LIN {X 103.200,Y -21.699,Z -137.911,A -90.000,B 90.000,C 0.000} C_DIS
LIN {X 103.154,Y -21.706,Z -138.831,A -90.000,B 90.000,C 0.000} C_DIS
LIN {X 102.985,Y -21.715,Z -141.880,A -90.000,B 90.000,C 0.000} C_DIS
LIN {X 102.956,Y -21.718,Z -142.349,A -90.000,B 90.000,C 0.000} C_DIS
LIN {X 102.711,Y -21.728,Z -146.129,A -90.000,B 90.000,C 0.000} C_DIS
LIN {X 102.478,Y -21.737,Z -149.340,A -90.000,B 90.000,C 0.000} C_DIS
LIN {X 102.272,Y -21.746,Z -151.898,A -90.000,B 90.000,C 0.000} C_DIS
LIN {X 102.195,Y -21.747,Z -152.952,A -90.000,B 90.000,C 0.000} C_DIS
LIN {X 102.172,Y -21.748,Z -153.237,A -90.000,B 90.000,C 0.000} C_DIS
LIN {X 101.990,Y -21.757,Z -155.321,A -90.000,B 90.000,C 0.000} C_DIS
LIN {X 101.952,Y -21.757,Z -155.803,A -90.000,B 90.000,C 0.000} C_DIS
LIN {X 101.875,Y -21.759,Z -156.808,A -90.000,B 90.000,C 0.000} C_DIS
LIN {X 101.833,Y -21.759,Z -157.268,A -90.000,B 90.000,C 0.000} C_DIS
LIN {X 101.694,Y -21.768,Z -158.747,A -90.000,B 90.000,C 0.000} C_DIS
LIN {X 101.636,Y -21.768,Z -159.458,A -90.000,B 90.000,C 0.000} C_DIS
LIN {X 101.552,Y -21.770,Z -160.519,A -90.000,B 90.000,C 0.000} C_DIS
LIN {X 101.526,Y -21.769,Z -160.801,A -90.000,B 90.000,C 0.000} C_DIS
LIN {X 101.473,Y -21.773,Z -161.328,A -90.000,B 90.000,C 0.000} C_DIS
LIN {X 101.406,Y -21.769,Z -162.061,A -90.000,B 90.000,C 0.000} C_DIS
LIN {X 101.227,Y -21.773,Z -164.255,A -90.000,B 90.000,C 0.000} C_DIS
LIN {X 101.195,Y -21.774,Z -164.609,A -90.000,B 90.000,C 0.000} C_DIS
LIN {X 101.168,Y -21.773,Z -164.885,A -90.000,B 90.000,C 0.000} C_DIS
LIN {X 100.874,Y -21.791,Z -168.265,A -90.000,B 90.000,C 0.000} C_DIS
LIN {X 100.554,Y -21.808,Z -171.701,A -90.000,B 90.000,C 0.000} C_DIS
LIN {X 100.400,Y -21.816,Z -173.250,A -90.000,B 90.000,C 0.000} C_DIS
LIN {X 100.226,Y -21.828,Z -174.986,A -90.000,B 90.000,C 0.000} C_DIS
LIN {X 100.198,Y -21.826,Z -175.266,A -90.000,B 90.000,C 0.000} C_DIS
LIN {X 99.941,Y -21.835,Z -177.681,A -90.000,B 90.000,C 0.000} C_DIS
LIN {X 99.892,Y -21.832,Z -178.165,A -90.000,B 90.000,C 0.000} C_DIS
LIN {X 99.862,Y -21.833,Z -178.432,A -90.000,B 90.000,C 0.000} C_DIS
LIN {X 99.723,Y -21.828,Z -179.586,A -90.000,B 90.000,C 0.000} C_DIS
LIN {X 99.550,Y -21.810,Z -181.085,A -90.000,B 90.000,C 0.000} C_DIS
LIN {X 99.434,Y -21.803,Z -182.000,A -90.000,B 90.000,C 0.000} C_DIS
LIN {X 99.202,Y -21.777,Z -183.867,A -90.000,B 90.000,C 0.000} C_DIS
LIN {X 99.146,Y -21.771,Z -184.282,A -90.000,B 90.000,C 0.000} C_DIS
LIN {X 98.820,Y -21.726,Z -186.729,A -90.000,B 90.000,C 0.000} C_DIS
LIN {X 98.551,Y -21.689,Z -188.733,A -90.000,B 90.000,C 0.000} C_DIS
LIN {X 98.240,Y -21.655,Z -191.111,A -90.000,B 90.000,C 0.000} C_DIS
LIN {X 98.078,Y -21.642,Z -192.230,A -90.000,B 90.000,C 0.000} C_DIS
LIN {X 97.900,Y -21.626,Z -193.439,A -90.000,B 90.000,C 0.000} C_DIS
LIN {X 97.865,Y -21.625,Z -193.671,A -90.000,B 90.000,C 0.000} C_DIS
LIN {X 97.839,Y -21.622,Z -193.828,A -90.000,B 90.000,C 0.000} C_DIS
LIN {X 97.584,Y -21.620,Z -195.289,A -90.000,B 90.000,C 0.000} C_DIS
LIN {X 97.330,Y -21.612,Z -196.692,A -90.000,B 90.000,C 0.000} C_DIS
LIN {X 97.302,Y -21.611,Z -196.843,A -90.000,B 90.000,C 0.000} C_DIS
LIN {X 97.260,Y -21.612,Z -197.057,A -90.000,B 90.000,C 0.000} C_DIS
LIN {X 96.796,Y -21.616,Z -199.323,A -90.000,B 90.000,C 0.000} C_DIS
LIN {X 96.529,Y -21.612,Z -200.569,A -90.000,B 90.000,C 0.000} C_DIS
LIN {X 96.463,Y -21.611,Z -200.859,A -90.000,B 90.000,C 0.000} C_DIS
LIN {X 95.804,Y -21.631,Z -203.660,A -90.000,B 90.000,C 0.000} C_DIS
LIN {X 95.494,Y -21.634,Z -204.941,A -90.000,B 90.000,C 0.000} C_DIS
LIN {X 95.323,Y -21.635,Z -205.637,A -90.000,B 90.000,C 0.000} C_DIS
LIN {X 94.278,Y -21.666,Z -209.816,A -90.000,B 90.000,C 0.000} C_DIS
LIN {X 93.985,Y -21.666,Z -210.965,A -90.000,B 90.000,C 0.000} C_DIS
LIN {X 92.877,Y -21.692,Z -215.251,A -90.000,B 90.000,C 0.000} C_DIS
LIN {X 92.712,Y -21.692,Z -215.887,A -90.000,B 90.000,C 0.000} C_DIS
LIN {X 92.490,Y -21.690,Z -216.750,A -90.000,B 90.000,C 0.000} C_DIS
LIN {X 91.455,Y -21.706,Z -220.703,A -90.000,B 90.000,C 0.000} C_DIS
LIN {X 90.619,Y -21.709,Z -223.906,A -90.000,B 90.000,C 0.000} C_DIS
LIN {X 90.094,Y -21.704,Z -225.931,A -90.000,B 90.000,C 0.000} C_DIS
LIN {X 90.051,Y -21.703,Z -226.091,A -90.000,B 90.000,C 0.000} C_DIS
LIN {X 89.413,Y -21.699,Z -228.410,A -90.000,B 90.000,C 0.000} C_DIS
LIN {X 88.561,Y -21.691,Z -231.519,A -90.000,B 90.000,C 0.000} C_DIS
LIN {X 88.509,Y -21.688,Z -231.694,A -90.000,B 90.000,C 0.000} C_DIS
LIN {X 87.993,Y -21.687,Z -233.408,A -90.000,B 90.000,C 0.000} C_DIS
LIN {X 86.773,Y -21.676,Z -237.465,A -90.000,B 90.000,C 0.000} C_DIS
LIN {X 86.686,Y -21.679,Z -237.741,A -90.000,B 90.000,C 0.000} C_DIS
LIN {X 86.213,Y -21.680,Z -239.140,A -90.000,B 90.000,C 0.000} C_DIS
LIN {X 85.045,Y -21.673,Z -242.614,A -90.000,B 90.000,C 0.000} C_DIS
LIN {X 84.730,Y -21.673,Z -243.561,A -90.000,B 90.000,C 0.000} C_DIS
LIN {X 84.730,Y -60.000,Z -243.561,A -90.000,B 90.000,C 0.000} C_DIS
LIN {X -106.254,Y -60.000,Z -243.561,A -90.000,B 90.000,C 0.000} C_DIS
LIN {X -106.254,Y -21.411,Z -243.561,A -90.000,B 90.000,C 0.000} C_DIS
LIN {X -105.827,Y -21.342,Z -243.259,A -90.000,B 90.000,C 0.000} C_DIS
LIN {X -103.067,Y -21.337,Z -241.434,A -90.000,B 90.000,C 0.000} C_DIS
LIN {X -99.700,Y -21.332,Z -239.239,A -90.000,B 90.000,C 0.000} C_DIS
LIN {X -95.248,Y -21.329,Z -236.322,A -90.000,B 90.000,C 0.000} C_DIS
LIN {X -91.046,Y -21.329,Z -233.611,A -90.000,B 90.000,C 0.000} C_DIS
LIN {X -87.083,Y -21.328,Z -231.061,A -90.000,B 90.000,C 0.000} C_DIS
LIN {X -82.491,Y -21.331,Z -228.162,A -90.000,B 90.000,C 0.000} C_DIS
LIN {X -81.014,Y -21.331,Z -227.236,A -90.000,B 90.000,C 0.000} C_DIS
LIN {X -78.594,Y -21.335,Z -225.697,A -90.000,B 90.000,C 0.000} C_DIS
LIN {X -73.982,Y -21.346,Z -222.839,A -90.000,B 90.000,C 0.000} C_DIS
LIN {X -71.749,Y -21.350,Z -221.468,A -90.000,B 90.000,C 0.000} C_DIS
LIN {X -69.686,Y -21.361,Z -220.171,A -90.000,B 90.000,C 0.000} C_DIS
LIN {X -66.193,Y -21.389,Z -217.992,A -90.000,B 90.000,C 0.000} C_DIS
LIN {X -62.248,Y -21.420,Z -215.563,A -90.000,B 90.000,C 0.000} C_DIS
LIN {X -59.889,Y -21.450,Z -214.098,A -90.000,B 90.000,C 0.000} C_DIS
LIN {X -57.151,Y -21.489,Z -212.404,A -90.000,B 90.000,C 0.000} C_DIS
LIN {X -54.976,Y -21.517,Z -211.076,A -90.000,B 90.000,C 0.000} C_DIS
LIN {X -54.531,Y -21.522,Z -210.805,A -90.000,B 90.000,C 0.000} C_DIS
LIN {X -53.089,Y -21.553,Z -209.900,A -90.000,B 90.000,C 0.000} C_DIS
LIN {X -52.244,Y -21.569,Z -209.368,A -90.000,B 90.000,C 0.000} C_DIS
LIN {X -49.132,Y -21.649,Z -207.418,A -90.000,B 90.000,C 0.000} C_DIS
LIN {X -47.972,Y -21.680,Z -206.695,A -90.000,B 90.000,C 0.000} C_DIS
LIN {X -46.144,Y -21.761,Z -205.510,A -90.000,B 90.000,C 0.000} C_DIS
LIN {X -43.428,Y -21.875,Z -203.761,A -90.000,B 90.000,C 0.000} C_DIS
LIN {X -42.555,Y -21.907,Z -203.192,A -90.000,B 90.000,C 0.000} C_DIS
LIN {X -40.956,Y -22.000,Z -202.120,A -90.000,B 90.000,C 0.000} C_DIS
LIN {X -40.168,Y -22.045,Z -201.596,A -90.000,B 90.000,C 0.000} C_DIS
LIN {X -38.826,Y -22.111,Z -200.682,A -90.000,B 90.000,C 0.000} C_DIS
LIN {X -38.138,Y -22.136,Z -200.199,A -90.000,B 90.000,C 0.000} C_DIS
LIN {X -37.944,Y -22.141,Z -200.056,A -90.000,B 90.000,C 0.000} C_DIS
LIN {X -37.389,Y -22.162,Z -199.640,A -90.000,B 90.000,C 0.000} C_DIS
LIN {X -36.329,Y -22.200,Z -198.837,A -90.000,B 90.000,C 0.000} C_DIS
LIN {X -34.180,Y -22.222,Z -197.104,A -90.000,B 90.000,C 0.000} C_DIS
LIN {X -33.953,Y -22.227,Z -196.919,A -90.000,B 90.000,C 0.000} C_DIS
LIN {X -32.090,Y -22.228,Z -195.331,A -90.000,B 90.000,C 0.000} C_DIS
LIN {X -30.755,Y -22.235,Z -194.205,A -90.000,B 90.000,C 0.000} C_DIS
LIN {X -30.074,Y -22.236,Z -193.626,A -90.000,B 90.000,C 0.000} C_DIS
LIN {X -27.945,Y -22.226,Z -191.825,A -90.000,B 90.000,C 0.000} C_DIS
LIN {X -27.695,Y -22.227,Z -191.609,A -90.000,B 90.000,C 0.000} C_DIS
LIN {X -27.149,Y -22.223,Z -191.131,A -90.000,B 90.000,C 0.000} C_DIS
LIN {X -25.105,Y -22.209,Z -189.370,A -90.000,B 90.000,C 0.000} C_DIS
LIN {X -24.930,Y -22.211,Z -189.215,A -90.000,B 90.000,C 0.000} C_DIS
LIN {X -24.541,Y -22.207,Z -188.853,A -90.000,B 90.000,C 0.000} C_DIS
LIN {X -22.451,Y -22.186,Z -186.958,A -90.000,B 90.000,C 0.000} C_DIS
LIN {X -22.349,Y -22.189,Z -186.862,A -90.000,B 90.000,C 0.000} C_DIS
LIN {X -21.597,Y -22.182,Z -186.102,A -90.000,B 90.000,C 0.000} C_DIS
LIN {X -19.952,Y -22.162,Z -184.488,A -90.000,B 90.000,C 0.000} C_DIS
LIN {X -19.814,Y -22.165,Z -184.348,A -90.000,B 90.000,C 0.000} C_DIS
LIN {X -18.083,Y -22.145,Z -182.471,A -90.000,B 90.000,C 0.000} C_DIS
LIN {X -17.843,Y -22.144,Z -182.206,A -90.000,B 90.000,C 0.000} C_DIS
LIN {X -17.415,Y -22.140,Z -181.731,A -90.000,B 90.000,C 0.000} C_DIS
LIN {X -17.370,Y -22.141,Z -181.681,A -90.000,B 90.000,C 0.000} C_DIS
LIN {X -15.624,Y -22.116,Z -179.571,A -90.000,B 90.000,C 0.000} C_DIS
LIN {X -15.250,Y -22.115,Z -179.111,A -90.000,B 90.000,C 0.000} C_DIS
LIN {X -15.094,Y -22.118,Z -178.911,A -90.000,B 90.000,C 0.000} C_DIS
LIN {X -13.181,Y -22.081,Z -176.292,A -90.000,B 90.000,C 0.000} C_DIS
LIN {X -13.050,Y -22.081,Z -176.110,A -90.000,B 90.000,C 0.000} C_DIS
LIN {X -12.917,Y -22.086,Z -175.919,A -90.000,B 90.000,C 0.000} C_DIS
LIN {X -11.259,Y -22.045,Z -173.288,A -90.000,B 90.000,C 0.000} C_DIS
LIN {X -11.080,Y -22.054,Z -172.984,A -90.000,B 90.000,C 0.000} C_DIS
LIN {X -11.024,Y -22.054,Z -172.881,A -90.000,B 90.000,C 0.000} C_DIS
LIN {X -9.686,Y -22.001,Z -170.299,A -90.000,B 90.000,C 0.000} C_DIS
LIN {X -9.547,Y -22.011,Z -170.002,A -90.000,B 90.000,C 0.000} C_DIS
LIN {X -8.642,Y -21.959,Z -167.714,A -90.000,B 90.000,C 0.000} C_DIS
LIN {X -8.538,Y -21.958,Z -167.438,A -90.000,B 90.000,C 0.000} C_DIS
LIN {X -8.445,Y -21.971,Z -167.158,A -90.000,B 90.000,C 0.000} C_DIS
LIN {X -8.313,Y -21.957,Z -166.630,A -90.000,B 90.000,C 0.000} C_DIS
LIN {X -7.867,Y -21.918,Z -164.877,A -90.000,B 90.000,C 0.000} C_DIS
LIN {X -7.834,Y -21.932,Z -164.681,A -90.000,B 90.000,C 0.000} C_DIS
LIN {X -7.719,Y -21.897,Z -163.007,A -90.000,B 90.000,C 0.000} C_DIS
LIN {X -7.727,Y -21.880,Z -162.907,A -90.000,B 90.000,C 0.000} C_DIS
LIN {X -7.905,Y -21.856,Z -162.077,A -90.000,B 90.000,C 0.000} C_DIS
LIN {X -7.916,Y -21.856,Z -162.021,A -90.000,B 90.000,C 0.000} C_DIS
LIN {X -7.996,Y -21.815,Z -161.796,A -90.000,B 90.000,C 0.000} C_DIS
LIN {X -8.060,Y -21.780,Z -161.607,A -90.000,B 90.000,C 0.000} C_DIS
LIN {X -8.241,Y -21.777,Z -161.247,A -90.000,B 90.000,C 0.000} C_DIS
LIN {X -8.444,Y -21.725,Z -160.934,A -90.000,B 90.000,C 0.000} C_DIS
LIN {X -8.526,Y -21.707,Z -160.802,A -90.000,B 90.000,C 0.000} C_DIS
LIN {X -8.552,Y -21.701,Z -160.759,A -90.000,B 90.000,C 0.000} C_DIS
LIN {X -8.873,Y -21.698,Z -160.372,A -90.000,B 90.000,C 0.000} C_DIS
LIN {X -8.932,Y -21.690,Z -160.309,A -90.000,B 90.000,C 0.000} C_DIS
LIN {X -9.104,Y -21.665,Z -160.116,A -90.000,B 90.000,C 0.000} C_DIS
LIN {X -9.212,Y -21.651,Z -159.991,A -90.000,B 90.000,C 0.000} C_DIS
LIN {X -9.330,Y -21.635,Z -159.850,A -90.000,B 90.000,C 0.000} C_DIS
LIN {X -9.669,Y -21.633,Z -159.535,A -90.000,B 90.000,C 0.000} C_DIS
LIN {X -9.815,Y -21.629,Z -159.394,A -90.000,B 90.000,C 0.000} C_DIS
LIN {X -10.168,Y -21.615,Z -159.041,A -90.000,B 90.000,C 0.000} C_DIS
LIN {X -10.408,Y -21.600,Z -158.806,A -90.000,B 90.000,C 0.000} C_DIS
LIN {X -11.277,Y -21.572,Z -158.006,A -90.000,B 90.000,C 0.000} C_DIS
LIN {X -11.496,Y -21.566,Z -157.804,A -90.000,B 90.000,C 0.000} C_DIS
LIN {X -11.881,Y -21.564,Z -157.468,A -90.000,B 90.000,C 0.000} C_DIS
LIN {X -13.335,Y -21.535,Z -156.177,A -90.000,B 90.000,C 0.000} C_DIS
LIN {X -13.574,Y -21.533,Z -155.965,A -90.000,B 90.000,C 0.000} C_DIS
LIN {X -15.277,Y -21.506,Z -154.485,A -90.000,B 90.000,C 0.000} C_DIS
LIN {X -15.775,Y -21.504,Z -154.059,A -90.000,B 90.000,C 0.000} C_DIS
LIN {X -17.794,Y -21.486,Z -152.333,A -90.000,B 90.000,C 0.000} C_DIS
LIN {X -18.467,Y -21.486,Z -151.758,A -90.000,B 90.000,C 0.000} C_DIS
LIN {X -20.638,Y -21.477,Z -149.908,A -90.000,B 90.000,C 0.000} C_DIS
LIN {X -20.734,Y -21.476,Z -149.825,A -90.000,B 90.000,C 0.000} C_DIS
LIN {X -20.875,Y -21.474,Z -149.698,A -90.000,B 90.000,C 0.000} C_DIS
LIN {X -23.951,Y -21.471,Z -146.908,A -90.000,B 90.000,C 0.000} C_DIS
LIN {X -24.114,Y -21.467,Z -146.745,A -90.000,B 90.000,C 0.000} C_DIS
LIN {X -27.216,Y -21.470,Z -143.581,A -90.000,B 90.000,C 0.000} C_DIS
LIN {X -27.540,Y -21.469,Z -143.244,A -90.000,B 90.000,C 0.000} C_DIS
LIN {X -27.679,Y -21.463,Z -143.078,A -90.000,B 90.000,C 0.000} C_DIS
LIN {X -29.860,Y -21.467,Z -140.414,A -90.000,B 90.000,C 0.000} C_DIS
LIN {X -30.541,Y -21.469,Z -139.579,A -90.000,B 90.000,C 0.000} C_DIS
LIN {X -30.827,Y -21.467,Z -139.209,A -90.000,B 90.000,C 0.000} C_DIS
LIN {X -31.012,Y -21.456,Z -138.921,A -90.000,B 90.000,C 0.000} C_DIS
LIN {X -32.519,Y -21.455,Z -136.513,A -90.000,B 90.000,C 0.000} C_DIS
LIN {X -33.305,Y -21.445,Z -135.260,A -90.000,B 90.000,C 0.000} C_DIS
LIN {X -33.469,Y -21.442,Z -134.995,A -90.000,B 90.000,C 0.000} C_DIS
LIN {X -33.552,Y -21.435,Z -134.865,A -90.000,B 90.000,C 0.000} C_DIS
LIN {X -33.811,Y -21.400,Z -134.386,A -90.000,B 90.000,C 0.000} C_DIS
LIN {X -34.144,Y -21.377,Z -133.751,A -90.000,B 90.000,C 0.000} C_DIS
LIN {X -34.605,Y -21.351,Z -132.868,A -90.000,B 90.000,C 0.000} C_DIS
LIN {X -35.010,Y -21.334,Z -132.094,A -90.000,B 90.000,C 0.000} C_DIS
LIN {X -35.479,Y -21.319,Z -131.192,A -90.000,B 90.000,C 0.000} C_DIS
LIN {X -35.801,Y -21.313,Z -130.570,A -90.000,B 90.000,C 0.000} C_DIS
LIN {X -35.993,Y -21.309,Z -130.154,A -90.000,B 90.000,C 0.000} C_DIS
LIN {X -36.367,Y -21.308,Z -129.339,A -90.000,B 90.000,C 0.000} C_DIS
LIN {X -36.397,Y -28.383,Z -129.274,A -90.000,B 90.000,C 0.000} C_DIS
LIN {X -36.412,Y -28.431,Z -129.242,A -90.000,B 90.000,C 0.000} C_DIS
LIN {X -36.426,Y -28.469,Z -129.210,A -90.000,B 90.000,C 0.000} C_DIS
LIN {X -36.482,Y -28.578,Z -129.090,A -90.000,B 90.000,C 0.000} C_DIS
LIN {X -36.582,Y -28.727,Z -128.872,A -90.000,B 90.000,C 0.000} C_DIS
LIN {X -36.744,Y -28.960,Z -128.520,A -90.000,B 90.000,C 0.000} C_DIS
LIN {X -36.860,Y -29.119,Z -128.269,A -90.000,B 90.000,C 0.000} C_DIS
LIN {X -36.940,Y -29.195,Z -128.101,A -90.000,B 90.000,C 0.000} C_DIS
LIN {X -36.990,Y -29.211,Z -128.000,A -90.000,B 90.000,C 0.000} C_DIS
LIN {X -37.006,Y -29.205,Z -127.970,A -90.000,B 90.000,C 0.000} C_DIS
LIN {X -37.018,Y -29.192,Z -127.950,A -90.000,B 90.000,C 0.000} C_DIS
LIN {X -37.027,Y -29.171,Z -127.939,A -90.000,B 90.000,C 0.000} C_DIS
LIN {X -37.033,Y -29.143,Z -127.934,A -90.000,B 90.000,C 0.000} C_DIS
LIN {X -37.038,Y -29.106,Z -127.933,A -90.000,B 90.000,C 0.000} C_DIS
LIN {X -37.054,Y -28.934,Z -127.937,A -90.000,B 90.000,C 0.000} C_DIS
LIN {X -37.063,Y -28.862,Z -127.934,A -90.000,B 90.000,C 0.000} C_DIS
LIN {X -37.076,Y -28.785,Z -127.924,A -90.000,B 90.000,C 0.000} C_DIS
LIN {X -37.093,Y -28.705,Z -127.907,A -90.000,B 90.000,C 0.000} C_DIS
LIN {X -37.116,Y -28.623,Z -127.880,A -90.000,B 90.000,C 0.000} C_DIS
LIN {X -37.145,Y -28.539,Z -127.841,A -90.000,B 90.000,C 0.000} C_DIS
LIN {X -37.227,Y -28.341,Z -127.718,A -90.000,B 90.000,C 0.000} C_DIS
LIN {X -37.282,Y -28.167,Z -127.630,A -90.000,B 90.000,C 0.000} C_DIS
LIN {X -37.347,Y -27.945,Z -127.522,A -90.000,B 90.000,C 0.000} C_DIS
LIN {X -37.424,Y -27.738,Z -127.391,A -90.000,B 90.000,C 0.000} C_DIS
LIN {X -37.467,Y -27.640,Z -127.317,A -90.000,B 90.000,C 0.000} C_DIS
LIN {X -37.513,Y -27.547,Z -127.237,A -90.000,B 90.000,C 0.000} C_DIS
LIN {X -37.616,Y -27.376,Z -127.055,A -90.000,B 90.000,C 0.000} C_DIS
LIN {X -37.733,Y -27.229,Z -126.846,A -90.000,B 90.000,C 0.000} C_DIS
LIN {X -37.865,Y -21.308,Z -126.605,A -90.000,B 90.000,C 0.000} C_DIS
LIN {X -37.912,Y -21.311,Z -126.520,A -90.000,B 90.000,C 0.000} C_DIS
LIN {X -38.002,Y -21.308,Z -126.356,A -90.000,B 90.000,C 0.000} C_DIS
LIN {X -38.241,Y -21.302,Z -125.917,A -90.000,B 90.000,C 0.000} C_DIS
LIN {X -38.627,Y -21.291,Z -125.197,A -90.000,B 90.000,C 0.000} C_DIS
LIN {X -38.777,Y -21.287,Z -124.909,A -90.000,B 90.000,C 0.000} C_DIS
LIN {X -39.004,Y -21.280,Z -124.458,A -90.000,B 90.000,C 0.000} C_DIS
LIN {X -39.147,Y -21.276,Z -124.151,A -90.000,B 90.000,C 0.000} C_DIS
LIN {X -39.192,Y -21.275,Z -124.043,A -90.000,B 90.000,C 0.000} C_DIS
LIN {X -39.222,Y -21.274,Z -123.959,A -90.000,B 90.000,C 0.000} C_DIS
LIN {X -39.240,Y -21.274,Z -123.897,A -90.000,B 90.000,C 0.000} C_DIS
LIN {X -39.247,Y -21.274,Z -123.853,A -90.000,B 90.000,C 0.000} C_DIS
LIN {X -39.248,Y -21.275,Z -123.837,A -90.000,B 90.000,C 0.000} C_DIS
LIN {X -39.243,Y -21.275,Z -123.814,A -90.000,B 90.000,C 0.000} C_DIS
LIN {X -39.231,Y -21.277,Z -123.796,A -90.000,B 90.000,C 0.000} C_DIS
LIN {X -39.229,Y -24.995,Z -123.795,A -90.000,B 90.000,C 0.000} C_DIS
LIN {X -39.214,Y -25.327,Z -123.786,A -90.000,B 90.000,C 0.000} C_DIS
LIN {X -39.195,Y -25.607,Z -123.774,A -90.000,B 90.000,C 0.000} C_DIS
LIN {X -39.190,Y -26.835,Z -123.768,A -90.000,B 90.000,C 0.000} C_DIS
LIN {X -39.184,Y -27.144,Z -123.749,A -90.000,B 90.000,C 0.000} C_DIS
LIN {X -39.183,Y -27.284,Z -123.737,A -90.000,B 90.000,C 0.000} C_DIS
LIN {X -39.184,Y -27.413,Z -123.721,A -90.000,B 90.000,C 0.000} C_DIS
LIN {X -39.187,Y -27.501,Z -123.701,A -90.000,B 90.000,C 0.000} C_DIS
LIN {X -39.193,Y -27.560,Z -123.678,A -90.000,B 90.000,C 0.000} C_DIS
LIN {X -39.201,Y -27.601,Z -123.650,A -90.000,B 90.000,C 0.000} C_DIS
LIN {X -39.213,Y -27.628,Z -123.617,A -90.000,B 90.000,C 0.000} C_DIS
LIN {X -39.227,Y -27.644,Z -123.579,A -90.000,B 90.000,C 0.000} C_DIS
LIN {X -39.245,Y -27.649,Z -123.535,A -90.000,B 90.000,C 0.000} C_DIS
LIN {X -39.293,Y -27.626,Z -123.427,A -90.000,B 90.000,C 0.000} C_DIS
LIN {X -39.358,Y -27.557,Z -123.292,A -90.000,B 90.000,C 0.000} C_DIS
LIN {X -39.442,Y -27.431,Z -123.124,A -90.000,B 90.000,C 0.000} C_DIS
LIN {X -39.548,Y -27.209,Z -122.920,A -90.000,B 90.000,C 0.000} C_DIS
LIN {X -39.609,Y -27.010,Z -122.804,A -90.000,B 90.000,C 0.000} C_DIS
LIN {X -39.677,Y -26.762,Z -122.677,A -90.000,B 90.000,C 0.000} C_DIS
LIN {X -39.832,Y -26.048,Z -122.392,A -90.000,B 90.000,C 0.000} C_DIS
LIN {X -39.920,Y -25.940,Z -122.232,A -90.000,B 90.000,C 0.000} C_DIS
LIN {X -40.015,Y -25.671,Z -122.059,A -90.000,B 90.000,C 0.000} C_DIS
LIN {X -40.117,Y -25.288,Z -121.875,A -90.000,B 90.000,C 0.000} C_DIS
LIN {X -40.228,Y -24.868,Z -121.677,A -90.000,B 90.000,C 0.000} C_DIS
LIN {X -40.286,Y -24.530,Z -121.573,A -90.000,B 90.000,C 0.000} C_DIS
LIN {X -40.346,Y -24.063,Z -121.466,A -90.000,B 90.000,C 0.000} C_DIS
LIN {X -40.472,Y -21.308,Z -121.241,A -90.000,B 90.000,C 0.000} C_DIS
LIN {X -40.603,Y -21.309,Z -121.009,A -90.000,B 90.000,C 0.000} C_DIS
LIN {X -41.229,Y -21.311,Z -119.874,A -90.000,B 90.000,C 0.000} C_DIS
LIN {X -41.474,Y -21.315,Z -119.505,A -90.000,B 90.000,C 0.000} C_DIS
LIN {X -41.800,Y -21.322,Z -118.973,A -90.000,B 90.000,C 0.000} C_DIS
LIN {X -41.907,Y -21.325,Z -118.798,A -90.000,B 90.000,C 0.000} C_DIS
LIN {X -42.253,Y -21.330,Z -118.234,A -90.000,B 90.000,C 0.000} C_DIS
LIN {X -42.719,Y -21.348,Z -117.601,A -90.000,B 90.000,C 0.000} C_DIS
LIN {X -42.949,Y -21.358,Z -117.266,A -90.000,B 90.000,C 0.000} C_DIS
LIN {X -43.532,Y -21.367,Z -116.420,A -90.000,B 90.000,C 0.000} C_DIS
LIN {X -43.898,Y -21.381,Z -115.938,A -90.000,B 90.000,C 0.000} C_DIS
LIN {X -44.128,Y -21.389,Z -115.633,A -90.000,B 90.000,C 0.000} C_DIS
LIN {X -44.279,Y -21.392,Z -115.432,A -90.000,B 90.000,C 0.000} C_DIS
LIN {X -45.329,Y -21.407,Z -114.023,A -90.000,B 90.000,C 0.000} C_DIS
LIN {X -45.721,Y -21.417,Z -113.518,A -90.000,B 90.000,C 0.000} C_DIS
LIN {X -45.896,Y -21.420,Z -113.288,A -90.000,B 90.000,C 0.000} C_DIS
LIN {X -46.606,Y -21.429,Z -112.363,A -90.000,B 90.000,C 0.000} C_DIS
LIN {X -47.556,Y -21.436,Z -111.104,A -90.000,B 90.000,C 0.000} C_DIS
LIN {X -48.722,Y -21.443,Z -109.567,A -90.000,B 90.000,C 0.000} C_DIS
LIN {X -49.146,Y -21.445,Z -109.011,A -90.000,B 90.000,C 0.000} C_DIS
LIN {X -50.156,Y -21.446,Z -107.700,A -90.000,B 90.000,C 0.000} C_DIS
LIN {X -50.687,Y -21.443,Z -106.997,A -90.000,B 90.000,C 0.000} C_DIS
LIN {X -50.978,Y -21.443,Z -106.620,A -90.000,B 90.000,C 0.000} C_DIS
LIN {X -51.545,Y -21.447,Z -105.883,A -90.000,B 90.000,C 0.000} C_DIS
LIN {X -52.480,Y -21.447,Z -104.644,A -90.000,B 90.000,C 0.000} C_DIS
LIN {X -52.745,Y -21.446,Z -104.304,A -90.000,B 90.000,C 0.000} C_DIS
LIN {X -53.236,Y -21.439,Z -103.643,A -90.000,B 90.000,C 0.000} C_DIS
LIN {X -53.973,Y -21.438,Z -102.642,A -90.000,B 90.000,C 0.000} C_DIS
LIN {X -54.159,Y -21.440,Z -102.398,A -90.000,B 90.000,C 0.000} C_DIS
LIN {X -55.294,Y -21.437,Z -100.911,A -90.000,B 90.000,C 0.000} C_DIS
LIN {X -55.652,Y -21.433,Z -100.429,A -90.000,B 90.000,C 0.000} C_DIS
LIN {X -56.207,Y -21.435,Z -99.698,A -90.000,B 90.000,C 0.000} C_DIS
LIN {X -57.185,Y -21.434,Z -98.372,A -90.000,B 90.000,C 0.000} C_DIS
LIN {X -57.678,Y -21.436,Z -97.725,A -90.000,B 90.000,C 0.000} C_DIS
LIN {X -58.066,Y -21.433,Z -97.206,A -90.000,B 90.000,C 0.000} C_DIS
LIN {X -58.754,Y -21.433,Z -96.281,A -90.000,B 90.000,C 0.000} C_DIS
LIN {X -59.071,Y -21.436,Z -95.868,A -90.000,B 90.000,C 0.000} C_DIS
LIN {X -60.236,Y -21.435,Z -94.352,A -90.000,B 90.000,C 0.000} C_DIS
LIN {X -60.305,Y -21.435,Z -94.261,A -90.000,B 90.000,C 0.000} C_DIS
LIN {X -61.166,Y -21.436,Z -93.167,A -90.000,B 90.000,C 0.000} C_DIS
LIN {X -61.831,Y -21.434,Z -92.297,A -90.000,B 90.000,C 0.000} C_DIS
LIN {X -62.049,Y -21.436,Z -92.021,A -90.000,B 90.000,C 0.000} C_DIS
LIN {X -62.501,Y -21.436,Z -91.470,A -90.000,B 90.000,C 0.000} C_DIS
LIN {X -63.781,Y -21.434,Z -89.886,A -90.000,B 90.000,C 0.000} C_DIS
LIN {X -64.037,Y -21.439,Z -89.589,A -90.000,B 90.000,C 0.000} C_DIS
LIN {X -64.811,Y -21.436,Z -88.698,A -90.000,B 90.000,C 0.000} C_DIS
LIN {X -65.500,Y -21.433,Z -87.889,A -90.000,B 90.000,C 0.000} C_DIS
LIN {X -65.849,Y -21.438,Z -87.501,A -90.000,B 90.000,C 0.000} C_DIS
LIN {X -67.254,Y -21.434,Z -85.954,A -90.000,B 90.000,C 0.000} C_DIS
LIN {X -67.768,Y -21.436,Z -85.403,A -90.000,B 90.000,C 0.000} C_DIS
LIN {X -68.995,Y -21.435,Z -84.081,A -90.000,B 90.000,C 0.000} C_DIS
LIN {X -69.616,Y -21.438,Z -83.426,A -90.000,B 90.000,C 0.000} C_DIS
LIN {X -70.059,Y -21.438,Z -82.958,A -90.000,B 90.000,C 0.000} C_DIS
LIN {X -70.778,Y -21.440,Z -82.196,A -90.000,B 90.000,C 0.000} C_DIS
LIN {X -71.040,Y -21.444,Z -81.928,A -90.000,B 90.000,C 0.000} C_DIS
LIN {X -72.383,Y -21.447,Z -80.558,A -90.000,B 90.000,C 0.000} C_DIS
LIN {X -72.753,Y -21.451,Z -80.201,A -90.000,B 90.000,C 0.000} C_DIS
LIN {X -73.384,Y -21.458,Z -79.594,A -90.000,B 90.000,C 0.000} C_DIS
LIN {X -73.817,Y -21.466,Z -79.186,A -90.000,B 90.000,C 0.000} C_DIS
LIN {X -74.097,Y -21.478,Z -78.942,A -90.000,B 90.000,C 0.000} C_DIS
LIN {X -74.657,Y -21.487,Z -78.466,A -90.000,B 90.000,C 0.000} C_DIS
LIN {X -74.749,Y -21.490,Z -78.391,A -90.000,B 90.000,C 0.000} C_DIS
LIN {X -75.018,Y -21.514,Z -78.215,A -90.000,B 90.000,C 0.000} C_DIS
LIN {X -75.134,Y -21.528,Z -78.147,A -90.000,B 90.000,C 0.000} C_DIS
LIN {X -75.214,Y -21.543,Z -78.117,A -90.000,B 90.000,C 0.000} C_DIS
LIN {X -75.475,Y -21.584,Z -78.023,A -90.000,B 90.000,C 0.000} C_DIS
LIN {X -75.630,Y -21.573,Z -77.985,A -90.000,B 90.000,C 0.000} C_DIS
LIN {X -75.665,Y -21.571,Z -77.978,A -90.000,B 90.000,C 0.000} C_DIS
LIN {X -75.962,Y -21.562,Z -77.935,A -90.000,B 90.000,C 0.000} C_DIS
LIN {X -76.435,Y -21.538,Z -77.881,A -90.000,B 90.000,C 0.000} C_DIS
LIN {X -76.793,Y -21.523,Z -77.836,A -90.000,B 90.000,C 0.000} C_DIS
LIN {X -76.898,Y -21.522,Z -77.823,A -90.000,B 90.000,C 0.000} C_DIS
LIN {X -77.125,Y -21.523,Z -77.791,A -90.000,B 90.000,C 0.000} C_DIS
LIN {X -77.349,Y -21.522,Z -77.754,A -90.000,B 90.000,C 0.000} C_DIS
LIN {X -77.592,Y -21.528,Z -77.711,A -90.000,B 90.000,C 0.000} C_DIS
LIN {X -78.198,Y -21.531,Z -77.557,A -90.000,B 90.000,C 0.000} C_DIS
LIN {X -78.441,Y -21.530,Z -77.494,A -90.000,B 90.000,C 0.000} C_DIS
LIN {X -78.826,Y -21.523,Z -77.382,A -90.000,B 90.000,C 0.000} C_DIS
LIN {X -79.214,Y -21.506,Z -77.239,A -90.000,B 90.000,C 0.000} C_DIS
LIN {X -79.342,Y -21.502,Z -77.191,A -90.000,B 90.000,C 0.000} C_DIS
LIN {X -79.680,Y -21.500,Z -77.061,A -90.000,B 90.000,C 0.000} C_DIS
LIN {X -80.183,Y -21.501,Z -76.863,A -90.000,B 90.000,C 0.000} C_DIS
LIN {X -80.384,Y -21.506,Z -76.780,A -90.000,B 90.000,C 0.000} C_DIS
LIN {X -80.558,Y -21.510,Z -76.701,A -90.000,B 90.000,C 0.000} C_DIS
LIN {X -80.720,Y -21.510,Z -76.620,A -90.000,B 90.000,C 0.000} C_DIS
LIN {X -81.147,Y -21.506,Z -76.395,A -90.000,B 90.000,C 0.000} C_DIS
LIN {X -81.483,Y -21.499,Z -76.201,A -90.000,B 90.000,C 0.000} C_DIS
LIN {X -82.494,Y -21.507,Z -75.604,A -90.000,B 90.000,C 0.000} C_DIS
LIN {X -82.881,Y -21.507,Z -75.343,A -90.000,B 90.000,C 0.000} C_DIS
LIN {X -83.072,Y -21.507,Z -75.209,A -90.000,B 90.000,C 0.000} C_DIS
LIN {X -84.075,Y -21.529,Z -74.451,A -90.000,B 90.000,C 0.000} C_DIS
LIN {X -84.524,Y -21.531,Z -74.071,A -90.000,B 90.000,C 0.000} C_DIS
LIN {X -84.785,Y -21.542,Z -73.841,A -90.000,B 90.000,C 0.000} C_DIS
LIN {X -85.413,Y -21.579,Z -73.276,A -90.000,B 90.000,C 0.000} C_DIS
LIN {X -85.548,Y -21.592,Z -73.165,A -90.000,B 90.000,C 0.000} C_DIS
LIN {X -85.783,Y -21.608,Z -72.952,A -90.000,B 90.000,C 0.000} C_DIS
LIN {X -85.872,Y -21.616,Z -72.870,A -90.000,B 90.000,C 0.000} C_DIS
LIN {X -86.020,Y -21.626,Z -72.728,A -90.000,B 90.000,C 0.000} C_DIS
LIN {X -86.245,Y -21.652,Z -72.505,A -90.000,B 90.000,C 0.000} C_DIS
LIN {X -86.681,Y -21.718,Z -72.085,A -90.000,B 90.000,C 0.000} C_DIS
LIN {X -87.118,Y -21.770,Z -71.700,A -90.000,B 90.000,C 0.000} C_DIS
LIN {X -87.288,Y -21.786,Z -71.554,A -90.000,B 90.000,C 0.000} C_DIS
LIN {X -87.408,Y -21.795,Z -71.448,A -90.000,B 90.000,C 0.000} C_DIS
LIN {X -87.582,Y -21.802,Z -71.298,A -90.000,B 90.000,C 0.000} C_DIS
LIN {X -87.965,Y -21.817,Z -70.950,A -90.000,B 90.000,C 0.000} C_DIS
LIN {X -88.130,Y -21.818,Z -70.804,A -90.000,B 90.000,C 0.000} C_DIS
LIN {X -88.265,Y -21.818,Z -70.678,A -90.000,B 90.000,C 0.000} C_DIS
LIN {X -88.585,Y -21.810,Z -70.365,A -90.000,B 90.000,C 0.000} C_DIS
LIN {X -88.782,Y -21.816,Z -70.173,A -90.000,B 90.000,C 0.000} C_DIS
LIN {X -88.856,Y -21.816,Z -70.103,A -90.000,B 90.000,C 0.000} C_DIS
LIN {X -89.139,Y -21.808,Z -69.820,A -90.000,B 90.000,C 0.000} C_DIS
LIN {X -89.245,Y -21.809,Z -69.712,A -90.000,B 90.000,C 0.000} C_DIS
LIN {X -89.495,Y -21.805,Z -69.467,A -90.000,B 90.000,C 0.000} C_DIS
LIN {X -89.673,Y -21.801,Z -69.290,A -90.000,B 90.000,C 0.000} C_DIS
LIN {X -90.157,Y -21.792,Z -68.829,A -90.000,B 90.000,C 0.000} C_DIS
LIN {X -90.241,Y -21.791,Z -68.752,A -90.000,B 90.000,C 0.000} C_DIS
LIN {X -90.757,Y -21.778,Z -68.291,A -90.000,B 90.000,C 0.000} C_DIS
LIN {X -90.792,Y -21.776,Z -68.262,A -90.000,B 90.000,C 0.000} C_DIS
LIN {X -91.256,Y -21.763,Z -67.888,A -90.000,B 90.000,C 0.000} C_DIS
LIN {X -91.449,Y -21.762,Z -67.738,A -90.000,B 90.000,C 0.000} C_DIS
LIN {X -92.277,Y -21.746,Z -67.104,A -90.000,B 90.000,C 0.000} C_DIS
LIN {X -93.006,Y -21.736,Z -66.548,A -90.000,B 90.000,C 0.000} C_DIS
LIN {X -93.462,Y -21.726,Z -66.192,A -90.000,B 90.000,C 0.000} C_DIS
LIN {X -93.961,Y -21.722,Z -65.795,A -90.000,B 90.000,C 0.000} C_DIS
LIN {X -94.235,Y -21.717,Z -65.575,A -90.000,B 90.000,C 0.000} C_DIS
LIN {X -94.480,Y -21.710,Z -65.370,A -90.000,B 90.000,C 0.000} C_DIS
LIN {X -95.101,Y -21.711,Z -64.837,A -90.000,B 90.000,C 0.000} C_DIS
LIN {X -95.412,Y -21.710,Z -64.565,A -90.000,B 90.000,C 0.000} C_DIS
LIN {X -96.015,Y -21.720,Z -64.029,A -90.000,B 90.000,C 0.000} C_DIS
LIN {X -96.780,Y -21.741,Z -63.356,A -90.000,B 90.000,C 0.000} C_DIS
LIN {X -97.028,Y -21.755,Z -63.146,A -90.000,B 90.000,C 0.000} C_DIS
LIN {X -97.383,Y -21.772,Z -62.848,A -90.000,B 90.000,C 0.000} C_DIS
LIN {X -97.482,Y -21.776,Z -62.763,A -90.000,B 90.000,C 0.000} C_DIS
LIN {X -97.976,Y -21.806,Z -62.362,A -90.000,B 90.000,C 0.000} C_DIS
LIN {X -98.434,Y -21.823,Z -62.000,A -90.000,B 90.000,C 0.000} C_DIS
LIN {X -98.556,Y -21.830,Z -61.905,A -90.000,B 90.000,C 0.000} C_DIS
LIN {X -99.011,Y -21.867,Z -61.535,A -90.000,B 90.000,C 0.000} C_DIS
LIN {X -99.479,Y -21.903,Z -61.149,A -90.000,B 90.000,C 0.000} C_DIS
LIN {X -99.549,Y -21.910,Z -61.088,A -90.000,B 90.000,C 0.000} C_DIS
LIN {X -99.908,Y -21.955,Z -60.767,A -90.000,B 90.000,C 0.000} C_DIS
LIN {X -100.184,Y -21.979,Z -60.501,A -90.000,B 90.000,C 0.000} C_DIS
LIN {X -100.513,Y -22.014,Z -60.175,A -90.000,B 90.000,C 0.000} C_DIS
LIN {X -100.696,Y -22.027,Z -59.987,A -90.000,B 90.000,C 0.000} C_DIS
LIN {X -100.973,Y -22.046,Z -59.692,A -90.000,B 90.000,C 0.000} C_DIS
LIN {X -101.017,Y -22.050,Z -59.643,A -90.000,B 90.000,C 0.000} C_DIS
LIN {X -101.358,Y -22.096,Z -59.245,A -90.000,B 90.000,C 0.000} C_DIS
LIN {X -101.602,Y -22.125,Z -58.947,A -90.000,B 90.000,C 0.000} C_DIS
LIN {X -101.659,Y -22.130,Z -58.868,A -90.000,B 90.000,C 0.000} C_DIS
LIN {X -102.004,Y -22.163,Z -58.362,A -90.000,B 90.000,C 0.000} C_DIS
LIN {X -102.079,Y -22.174,Z -58.245,A -90.000,B 90.000,C 0.000} C_DIS
LIN {X -102.241,Y -22.195,Z -57.967,A -90.000,B 90.000,C 0.000} C_DIS
LIN {X -102.421,Y -22.216,Z -57.648,A -90.000,B 90.000,C 0.000} C_DIS
LIN {X -102.455,Y -22.218,Z -57.583,A -90.000,B 90.000,C 0.000} C_DIS
LIN {X -102.526,Y -22.226,Z -57.437,A -90.000,B 90.000,C 0.000} C_DIS
LIN {X -102.651,Y -22.249,Z -57.154,A -90.000,B 90.000,C 0.000} C_DIS
LIN {X -102.783,Y -22.268,Z -56.845,A -90.000,B 90.000,C 0.000} C_DIS
LIN {X -102.885,Y -22.281,Z -56.599,A -90.000,B 90.000,C 0.000} C_DIS
LIN {X -102.989,Y -22.301,Z -56.321,A -90.000,B 90.000,C 0.000} C_DIS
LIN {X -103.015,Y -22.302,Z -56.245,A -90.000,B 90.000,C 0.000} C_DIS
LIN {X -103.058,Y -22.307,Z -56.102,A -90.000,B 90.000,C 0.000} C_DIS
LIN {X -103.208,Y -22.335,Z -55.521,A -90.000,B 90.000,C 0.000} C_DIS
LIN {X -103.249,Y -22.343,Z -55.348,A -90.000,B 90.000,C 0.000} C_DIS
LIN {X -103.268,Y -22.349,Z -55.258,A -90.000,B 90.000,C 0.000} C_DIS
LIN {X -103.303,Y -22.353,Z -55.050,A -90.000,B 90.000,C 0.000} C_DIS
LIN {X -103.359,Y -22.368,Z -54.628,A -90.000,B 90.000,C 0.000} C_DIS
LIN {X -103.366,Y -22.370,Z -54.559,A -90.000,B 90.000,C 0.000} C_DIS
LIN {X -103.395,Y -22.383,Z -54.228,A -90.000,B 90.000,C 0.000} C_DIS
LIN {X -103.400,Y -22.387,Z -54.048,A -90.000,B 90.000,C 0.000} C_DIS
LIN {X -103.397,Y -22.393,Z -53.898,A -90.000,B 90.000,C 0.000} C_DIS
LIN {X -103.372,Y -22.409,Z -53.538,A -90.000,B 90.000,C 0.000} C_DIS
LIN {X -103.355,Y -22.415,Z -53.337,A -90.000,B 90.000,C 0.000} C_DIS
LIN {X -103.330,Y -22.423,Z -53.067,A -90.000,B 90.000,C 0.000} C_DIS
LIN {X -103.322,Y -22.424,Z -53.016,A -90.000,B 90.000,C 0.000} C_DIS
LIN {X -103.297,Y -22.431,Z -52.884,A -90.000,B 90.000,C 0.000} C_DIS
LIN {X -103.272,Y -22.438,Z -52.768,A -90.000,B 90.000,C 0.000} C_DIS
LIN {X -103.224,Y -22.440,Z -52.576,A -90.000,B 90.000,C 0.000} C_DIS
LIN {X -103.184,Y -22.444,Z -52.436,A -90.000,B 90.000,C 0.000} C_DIS
LIN {X -103.160,Y -22.447,Z -52.365,A -90.000,B 90.000,C 0.000} C_DIS
LIN {X -103.202,Y -22.416,Z -52.282,A -90.000,B 90.000,C 0.000} C_DIS
LIN {X -103.424,Y -22.248,Z -51.790,A -90.000,B 90.000,C 0.000} C_DIS
LIN {X -103.504,Y -22.175,Z -51.587,A -90.000,B 90.000,C 0.000} C_DIS
LIN {X -103.624,Y -22.059,Z -51.259,A -90.000,B 90.000,C 0.000} C_DIS
LIN {X -103.723,Y -21.932,Z -50.918,A -90.000,B 90.000,C 0.000} C_DIS
LIN {X -103.756,Y -21.886,Z -50.789,A -90.000,B 90.000,C 0.000} C_DIS
LIN {X -103.779,Y -21.838,Z -50.656,A -90.000,B 90.000,C 0.000} C_DIS
LIN {X -103.789,Y -21.812,Z -50.581,A -90.000,B 90.000,C 0.000} C_DIS
LIN {X -103.972,Y -21.836,Z -50.313,A -90.000,B 90.000,C 0.000} C_DIS
LIN {X -104.139,Y -21.850,Z -50.053,A -90.000,B 90.000,C 0.000} C_DIS
LIN {X -104.320,Y -21.864,Z -49.755,A -90.000,B 90.000,C 0.000} C_DIS
LIN {X -104.581,Y -21.889,Z -49.318,A -90.000,B 90.000,C 0.000} C_DIS
LIN {X -104.642,Y -21.897,Z -49.208,A -90.000,B 90.000,C 0.000} C_DIS
LIN {X -104.735,Y -21.916,Z -49.021,A -90.000,B 90.000,C 0.000} C_DIS
LIN {X -104.846,Y -21.942,Z -48.793,A -90.000,B 90.000,C 0.000} C_DIS
LIN {X -105.092,Y -21.990,Z -48.229,A -90.000,B 90.000,C 0.000} C_DIS
LIN {X -105.136,Y -22.003,Z -48.120,A -90.000,B 90.000,C 0.000} C_DIS
LIN {X -105.277,Y -22.057,Z -47.703,A -90.000,B 90.000,C 0.000} C_DIS
LIN {X -105.376,Y -22.094,Z -47.352,A -90.000,B 90.000,C 0.000} C_DIS
LIN {X -105.462,Y -22.123,Z -47.005,A -90.000,B 90.000,C 0.000} C_DIS
LIN {X -105.501,Y -22.133,Z -46.825,A -90.000,B 90.000,C 0.000} C_DIS
LIN {X -105.526,Y -22.142,Z -46.692,A -90.000,B 90.000,C 0.000} C_DIS
LIN {X -105.541,Y -22.153,Z -46.588,A -90.000,B 90.000,C 0.000} C_DIS
LIN {X -105.582,Y -22.183,Z -46.213,A -90.000,B 90.000,C 0.000} C_DIS
LIN {X -105.591,Y -22.193,Z -46.119,A -90.000,B 90.000,C 0.000} C_DIS
LIN {X -105.608,Y -22.212,Z -45.853,A -90.000,B 90.000,C 0.000} C_DIS
LIN {X -105.612,Y -22.219,Z -45.761,A -90.000,B 90.000,C 0.000} C_DIS
LIN {X -105.604,Y -22.248,Z -45.415,A -90.000,B 90.000,C 0.000} C_DIS
LIN {X -105.599,Y -22.252,Z -45.328,A -90.000,B 90.000,C 0.000} C_DIS
LIN {X -105.589,Y -22.258,Z -45.213,A -90.000,B 90.000,C 0.000} C_DIS
LIN {X -105.559,Y -22.277,Z -44.943,A -90.000,B 90.000,C 0.000} C_DIS
LIN {X -105.529,Y -22.296,Z -44.717,A -90.000,B 90.000,C 0.000} C_DIS
LIN {X -105.503,Y -22.304,Z -44.548,A -90.000,B 90.000,C 0.000} C_DIS
LIN {X -105.470,Y -22.316,Z -44.388,A -90.000,B 90.000,C 0.000} C_DIS
LIN {X -105.409,Y -22.325,Z -44.126,A -90.000,B 90.000,C 0.000} C_DIS
LIN {X -105.393,Y -22.328,Z -44.068,A -90.000,B 90.000,C 0.000} C_DIS
LIN {X -105.336,Y -22.338,Z -43.897,A -90.000,B 90.000,C 0.000} C_DIS
LIN {X -105.283,Y -22.349,Z -43.748,A -90.000,B 90.000,C 0.000} C_DIS
LIN {X -105.213,Y -22.352,Z -43.572,A -90.000,B 90.000,C 0.000} C_DIS
LIN {X -105.082,Y -22.358,Z -43.258,A -90.000,B 90.000,C 0.000} C_DIS
LIN {X -105.019,Y -22.365,Z -43.126,A -90.000,B 90.000,C 0.000} C_DIS
LIN {X -104.842,Y -22.372,Z -42.834,A -90.000,B 90.000,C 0.000} C_DIS
LIN {X -104.659,Y -22.379,Z -42.541,A -90.000,B 90.000,C 0.000} C_DIS
LIN {X -104.607,Y -22.375,Z -42.463,A -90.000,B 90.000,C 0.000} C_DIS
LIN {X -104.531,Y -22.373,Z -42.356,A -90.000,B 90.000,C 0.000} C_DIS
LIN {X -104.452,Y -22.375,Z -42.257,A -90.000,B 90.000,C 0.000} C_DIS
LIN {X -104.222,Y -22.382,Z -41.988,A -90.000,B 90.000,C 0.000} C_DIS
LIN {X -103.968,Y -22.372,Z -41.717,A -90.000,B 90.000,C 0.000} C_DIS
LIN {X -103.928,Y -22.369,Z -41.676,A -90.000,B 90.000,C 0.000} C_DIS
LIN {X -103.793,Y -22.365,Z -41.553,A -90.000,B 90.000,C 0.000} C_DIS
LIN {X -103.705,Y -22.367,Z -41.479,A -90.000,B 90.000,C 0.000} C_DIS
LIN {X -103.482,Y -22.359,Z -41.299,A -90.000,B 90.000,C 0.000} C_DIS
LIN {X -103.433,Y -22.359,Z -41.263,A -90.000,B 90.000,C 0.000} C_DIS
LIN {X -103.155,Y -22.338,Z -41.076,A -90.000,B 90.000,C 0.000} C_DIS
LIN {X -103.027,Y -22.329,Z -40.992,A -90.000,B 90.000,C 0.000} C_DIS
LIN {X -102.803,Y -22.319,Z -40.854,A -90.000,B 90.000,C 0.000} C_DIS
LIN {X -102.747,Y -22.312,Z -40.822,A -90.000,B 90.000,C 0.000} C_DIS
LIN {X -102.620,Y -22.300,Z -40.756,A -90.000,B 90.000,C 0.000} C_DIS
LIN {X -102.435,Y -22.285,Z -40.667,A -90.000,B 90.000,C 0.000} C_DIS
LIN {X -102.287,Y -22.265,Z -40.601,A -90.000,B 90.000,C 0.000} C_DIS
LIN {X -102.209,Y -22.256,Z -40.569,A -90.000,B 90.000,C 0.000} C_DIS
LIN {X -101.720,Y -22.211,Z -40.390,A -90.000,B 90.000,C 0.000} C_DIS
LIN {X -101.487,Y -22.193,Z -40.314,A -90.000,B 90.000,C 0.000} C_DIS
LIN {X -101.404,Y -22.187,Z -40.288,A -90.000,B 90.000,C 0.000} C_DIS
LIN {X -101.283,Y -22.170,Z -40.256,A -90.000,B 90.000,C 0.000} C_DIS
LIN {X -101.182,Y -22.156,Z -40.232,A -90.000,B 90.000,C 0.000} C_DIS
LIN {X -101.098,Y -22.148,Z -40.216,A -90.000,B 90.000,C 0.000} C_DIS
LIN {X -100.666,Y -22.116,Z -40.146,A -90.000,B 90.000,C 0.000} C_DIS
LIN {X -100.488,Y -22.106,Z -40.124,A -90.000,B 90.000,C 0.000} C_DIS
LIN {X -99.958,Y -22.074,Z -40.065,A -90.000,B 90.000,C 0.000} C_DIS
LIN {X -99.681,Y -22.051,Z -40.042,A -90.000,B 90.000,C 0.000} C_DIS
LIN {X -99.430,Y -22.107,Z -39.965,A -90.000,B 90.000,C 0.000} C_DIS
LIN {X -99.290,Y -22.139,Z -39.928,A -90.000,B 90.000,C 0.000} C_DIS
LIN {X -99.046,Y -22.200,Z -39.866,A -90.000,B 90.000,C 0.000} C_DIS
LIN {X -98.902,Y -22.234,Z -39.835,A -90.000,B 90.000,C 0.000} C_DIS
LIN {X -98.578,Y -22.315,Z -39.782,A -90.000,B 90.000,C 0.000} C_DIS
LIN {X -98.212,Y -22.417,Z -39.729,A -90.000,B 90.000,C 0.000} C_DIS
LIN {X -97.944,Y -22.493,Z -39.698,A -90.000,B 90.000,C 0.000} C_DIS
LIN {X -97.572,Y -22.590,Z -39.665,A -90.000,B 90.000,C 0.000} C_DIS
LIN {X -97.478,Y -22.615,Z -39.660,A -90.000,B 90.000,C 0.000} C_DIS
LIN {X -97.260,Y -22.669,Z -39.655,A -90.000,B 90.000,C 0.000} C_DIS
LIN {X -96.838,Y -22.647,Z -39.160,A -90.000,B 90.000,C 0.000} C_DIS
LIN {X -96.756,Y -22.641,Z -39.046,A -90.000,B 90.000,C 0.000} C_DIS
LIN {X -96.658,Y -22.629,Z -38.931,A -90.000,B 90.000,C 0.000} C_DIS
LIN {X -96.388,Y -22.608,Z -38.652,A -90.000,B 90.000,C 0.000} C_DIS
LIN {X -96.165,Y -22.602,Z -38.428,A -90.000,B 90.000,C 0.000} C_DIS
LIN {X -96.043,Y -22.587,Z -38.282,A -90.000,B 90.000,C 0.000} C_DIS
LIN {X -95.769,Y -22.567,Z -37.998,A -90.000,B 90.000,C 0.000} C_DIS
LIN {X -95.651,Y -22.558,Z -37.889,A -90.000,B 90.000,C 0.000} C_DIS
LIN {X -95.361,Y -22.548,Z -37.639,A -90.000,B 90.000,C 0.000} C_DIS
LIN {X -95.110,Y -22.530,Z -37.391,A -90.000,B 90.000,C 0.000} C_DIS
LIN {X -95.048,Y -22.521,Z -37.332,A -90.000,B 90.000,C 0.000} C_DIS
LIN {X -94.966,Y -22.513,Z -37.257,A -90.000,B 90.000,C 0.000} C_DIS
LIN {X -94.896,Y -22.507,Z -37.200,A -90.000,B 90.000,C 0.000} C_DIS
LIN {X -94.604,Y -22.486,Z -36.969,A -90.000,B 90.000,C 0.000} C_DIS
LIN {X -94.544,Y -22.486,Z -36.919,A -90.000,B 90.000,C 0.000} C_DIS
LIN {X -94.317,Y -22.469,Z -36.742,A -90.000,B 90.000,C 0.000} C_DIS
LIN {X -93.967,Y -22.449,Z -36.512,A -90.000,B 90.000,C 0.000} C_DIS
LIN {X -93.948,Y -22.448,Z -36.499,A -90.000,B 90.000,C 0.000} C_DIS
LIN {X -93.729,Y -22.430,Z -36.326,A -90.000,B 90.000,C 0.000} C_DIS
LIN {X -93.620,Y -22.419,Z -36.248,A -90.000,B 90.000,C 0.000} C_DIS
LIN {X -93.494,Y -22.412,Z -36.169,A -90.000,B 90.000,C 0.000} C_DIS
LIN {X -93.249,Y -22.403,Z -36.028,A -90.000,B 90.000,C 0.000} C_DIS
LIN {X -93.104,Y -22.401,Z -35.946,A -90.000,B 90.000,C 0.000} C_DIS
LIN {X -92.947,Y -22.389,Z -35.838,A -90.000,B 90.000,C 0.000} C_DIS
LIN {X -92.809,Y -22.382,Z -35.750,A -90.000,B 90.000,C 0.000} C_DIS
LIN {X -92.626,Y -22.375,Z -35.645,A -90.000,B 90.000,C 0.000} C_DIS
LIN {X -92.532,Y -22.371,Z -35.591,A -90.000,B 90.000,C 0.000} C_DIS
LIN {X -92.405,Y -22.367,Z -35.524,A -90.000,B 90.000,C 0.000} C_DIS
LIN {X -92.257,Y -22.366,Z -35.451,A -90.000,B 90.000,C 0.000} C_DIS
LIN {X -91.902,Y -22.355,Z -35.250,A -90.000,B 90.000,C 0.000} C_DIS
LIN {X -91.783,Y -22.425,Z -35.139,A -90.000,B 90.000,C 0.000} C_DIS
LIN {X -91.713,Y -22.464,Z -35.081,A -90.000,B 90.000,C 0.000} C_DIS
LIN {X -91.494,Y -22.577,Z -34.921,A -90.000,B 90.000,C 0.000} C_DIS
LIN {X -91.304,Y -22.673,Z -34.790,A -90.000,B 90.000,C 0.000} C_DIS
LIN {X -91.202,Y -22.722,Z -34.723,A -90.000,B 90.000,C 0.000} C_DIS
LIN {X -91.120,Y -22.764,Z -34.661,A -90.000,B 90.000,C 0.000} C_DIS
LIN {X -90.995,Y -22.808,Z -34.578,A -90.000,B 90.000,C 0.000} C_DIS
LIN {X -90.835,Y -22.865,Z -34.476,A -90.000,B 90.000,C 0.000} C_DIS
LIN {X -90.844,Y -22.872,Z -34.379,A -90.000,B 90.000,C 0.000} C_DIS
LIN {X -90.861,Y -22.888,Z -34.147,A -90.000,B 90.000,C 0.000} C_DIS
LIN {X -90.865,Y -22.897,Z -34.016,A -90.000,B 90.000,C 0.000} C_DIS
LIN {X -90.863,Y -22.903,Z -33.945,A -90.000,B 90.000,C 0.000} C_DIS
LIN {X -90.855,Y -22.914,Z -33.828,A -90.000,B 90.000,C 0.000} C_DIS
LIN {X -90.864,Y -22.929,Z -33.597,A -90.000,B 90.000,C 0.000} C_DIS
LIN {X -90.869,Y -22.935,Z -33.369,A -90.000,B 90.000,C 0.000} C_DIS
LIN {X -90.865,Y -22.935,Z -33.276,A -90.000,B 90.000,C 0.000} C_DIS
LIN {X -90.843,Y -22.936,Z -33.080,A -90.000,B 90.000,C 0.000} C_DIS
LIN {X -90.823,Y -22.937,Z -32.977,A -90.000,B 90.000,C 0.000} C_DIS
LIN {X -90.785,Y -22.939,Z -32.802,A -90.000,B 90.000,C 0.000} C_DIS
LIN {X -90.753,Y -22.941,Z -32.677,A -90.000,B 90.000,C 0.000} C_DIS
LIN {X -90.735,Y -22.943,Z -32.619,A -90.000,B 90.000,C 0.000} C_DIS
LIN {X -90.703,Y -22.947,Z -32.527,A -90.000,B 90.000,C 0.000} C_DIS
LIN {X -90.676,Y -22.949,Z -32.459,A -90.000,B 90.000,C 0.000} C_DIS
LIN {X -90.618,Y -22.952,Z -32.333,A -90.000,B 90.000,C 0.000} C_DIS
LIN {X -90.575,Y -22.955,Z -32.251,A -90.000,B 90.000,C 0.000} C_DIS
LIN {X -90.511,Y -22.955,Z -32.133,A -90.000,B 90.000,C 0.000} C_DIS
LIN {X -90.460,Y -22.955,Z -32.044,A -90.000,B 90.000,C 0.000} C_DIS
LIN {X -90.426,Y -22.955,Z -31.991,A -90.000,B 90.000,C 0.000} C_DIS
LIN {X -90.240,Y -22.958,Z -31.750,A -90.000,B 90.000,C 0.000} C_DIS
LIN {X -89.910,Y -22.973,Z -31.385,A -90.000,B 90.000,C 0.000} C_DIS
LIN {X -89.771,Y -22.970,Z -31.206,A -90.000,B 90.000,C 0.000} C_DIS
LIN {X -89.672,Y -22.962,Z -31.083,A -90.000,B 90.000,C 0.000} C_DIS
LIN {X -89.641,Y -22.960,Z -31.047,A -90.000,B 90.000,C 0.000} C_DIS
LIN {X -89.549,Y -22.955,Z -30.950,A -90.000,B 90.000,C 0.000} C_DIS
LIN {X -89.436,Y -22.949,Z -30.836,A -90.000,B 90.000,C 0.000} C_DIS
LIN {X -89.366,Y -22.946,Z -30.769,A -90.000,B 90.000,C 0.000} C_DIS
LIN {X -89.271,Y -22.938,Z -30.689,A -90.000,B 90.000,C 0.000} C_DIS
LIN {X -89.161,Y -22.932,Z -30.607,A -90.000,B 90.000,C 0.000} C_DIS
LIN {X -89.052,Y -22.927,Z -30.537,A -90.000,B 90.000,C 0.000} C_DIS
LIN {X -88.818,Y -22.919,Z -30.398,A -90.000,B 90.000,C 0.000} C_DIS
LIN {X -88.654,Y -22.915,Z -30.305,A -90.000,B 90.000,C 0.000} C_DIS
LIN {X -88.340,Y -22.907,Z -30.165,A -90.000,B 90.000,C 0.000} C_DIS
LIN {X -88.256,Y -22.909,Z -30.134,A -90.000,B 90.000,C 0.000} C_DIS
LIN {X -87.918,Y -22.901,Z -29.997,A -90.000,B 90.000,C 0.000} C_DIS
LIN {X -87.947,Y -22.878,Z -29.887,A -90.000,B 90.000,C 0.000} C_DIS
LIN {X -87.973,Y -22.853,Z -29.763,A -90.000,B 90.000,C 0.000} C_DIS
LIN {X -87.985,Y -22.824,Z -29.661,A -90.000,B 90.000,C 0.000} C_DIS
LIN {X -87.995,Y -22.814,Z -29.591,A -90.000,B 90.000,C 0.000} C_DIS
LIN {X -88.010,Y -22.793,Z -29.497,A -90.000,B 90.000,C 0.000} C_DIS
LIN {X -88.021,Y -22.784,Z -29.431,A -90.000,B 90.000,C 0.000} C_DIS
LIN {X -88.039,Y -22.760,Z -29.253,A -90.000,B 90.000,C 0.000} C_DIS
LIN {X -88.062,Y -22.735,Z -29.011,A -90.000,B 90.000,C 0.000} C_DIS
LIN {X -88.060,Y -22.707,Z -28.813,A -90.000,B 90.000,C 0.000} C_DIS
LIN {X -88.057,Y -22.700,Z -28.765,A -90.000,B 90.000,C 0.000} C_DIS
LIN {X -88.046,Y -22.687,Z -28.677,A -90.000,B 90.000,C 0.000} C_DIS
LIN {X -88.011,Y -22.650,Z -28.406,A -90.000,B 90.000,C 0.000} C_DIS
LIN {X -87.985,Y -22.629,Z -28.271,A -90.000,B 90.000,C 0.000} C_DIS
LIN {X -87.964,Y -22.620,Z -28.171,A -90.000,B 90.000,C 0.000} C_DIS
LIN {X -87.931,Y -22.602,Z -28.050,A -90.000,B 90.000,C 0.000} C_DIS
LIN {X -87.900,Y -22.588,Z -27.949,A -90.000,B 90.000,C 0.000} C_DIS
LIN {X -87.753,Y -22.525,Z -27.543,A -90.000,B 90.000,C 0.000} C_DIS
LIN {X -87.729,Y -22.514,Z -27.482,A -90.000,B 90.000,C 0.000} C_DIS
LIN {X -87.672,Y -22.494,Z -27.349,A -90.000,B 90.000,C 0.000} C_DIS
LIN {X -87.535,Y -22.441,Z -27.083,A -90.000,B 90.000,C 0.000} C_DIS
LIN {X -87.498,Y -22.429,Z -27.015,A -90.000,B 90.000,C 0.000} C_DIS
LIN {X -87.441,Y -22.413,Z -26.919,A -90.000,B 90.000,C 0.000} C_DIS
LIN {X -87.306,Y -22.381,Z -26.702,A -90.000,B 90.000,C 0.000} C_DIS
LIN {X -87.236,Y -22.361,Z -26.594,A -90.000,B 90.000,C 0.000} C_DIS
LIN {X -87.140,Y -22.338,Z -26.453,A -90.000,B 90.000,C 0.000} C_DIS
LIN {X -86.929,Y -22.291,Z -26.173,A -90.000,B 90.000,C 0.000} C_DIS
LIN {X -86.869,Y -22.280,Z -26.096,A -90.000,B 90.000,C 0.000} C_DIS
LIN {X -86.481,Y -22.219,Z -25.623,A -90.000,B 90.000,C 0.000} C_DIS
LIN {X -86.423,Y -22.208,Z -25.555,A -90.000,B 90.000,C 0.000} C_DIS
LIN {X -86.186,Y -22.166,Z -25.287,A -90.000,B 90.000,C 0.000} C_DIS
LIN {X -85.862,Y -22.134,Z -24.949,A -90.000,B 90.000,C 0.000} C_DIS
LIN {X -85.723,Y -22.127,Z -24.811,A -90.000,B 90.000,C 0.000} C_DIS
LIN {X -85.224,Y -22.106,Z -24.319,A -90.000,B 90.000,C 0.000} C_DIS
LIN {X -85.084,Y -22.108,Z -24.180,A -90.000,B 90.000,C 0.000} C_DIS
LIN {X -84.541,Y -22.122,Z -23.645,A -90.000,B 90.000,C 0.000} C_DIS
LIN {X -83.949,Y -22.147,Z -23.067,A -90.000,B 90.000,C 0.000} C_DIS
LIN {X -83.851,Y -22.153,Z -22.969,A -90.000,B 90.000,C 0.000} C_DIS
LIN {X -83.737,Y -22.164,Z -22.860,A -90.000,B 90.000,C 0.000} C_DIS
LIN {X -83.426,Y -22.186,Z -22.580,A -90.000,B 90.000,C 0.000} C_DIS
LIN {X -83.182,Y -22.205,Z -22.371,A -90.000,B 90.000,C 0.000} C_DIS
LIN {X -82.987,Y -22.214,Z -22.211,A -90.000,B 90.000,C 0.000} C_DIS
LIN {X -82.867,Y -22.223,Z -22.116,A -90.000,B 90.000,C 0.000} C_DIS
LIN {X -82.600,Y -22.248,Z -21.916,A -90.000,B 90.000,C 0.000} C_DIS
LIN {X -82.500,Y -22.259,Z -21.845,A -90.000,B 90.000,C 0.000} C_DIS
LIN {X -82.236,Y -22.284,Z -21.669,A -90.000,B 90.000,C 0.000} C_DIS
LIN {X -82.100,Y -22.301,Z -21.585,A -90.000,B 90.000,C 0.000} C_DIS
LIN {X -81.721,Y -22.327,Z -21.372,A -90.000,B 90.000,C 0.000} C_DIS
LIN {X -81.327,Y -22.337,Z -21.180,A -90.000,B 90.000,C 0.000} C_DIS
LIN {X -81.087,Y -22.348,Z -21.075,A -90.000,B 90.000,C 0.000} C_DIS
LIN {X -80.920,Y -22.360,Z -21.009,A -90.000,B 90.000,C 0.000} C_DIS
LIN {X -80.831,Y -22.369,Z -20.978,A -90.000,B 90.000,C 0.000} C_DIS
LIN {X -80.728,Y -22.379,Z -20.946,A -90.000,B 90.000,C 0.000} C_DIS
LIN {X -80.337,Y -22.402,Z -20.843,A -90.000,B 90.000,C 0.000} C_DIS
LIN {X -80.280,Y -22.404,Z -20.829,A -90.000,B 90.000,C 0.000} C_DIS
LIN {X -80.066,Y -22.408,Z -20.790,A -90.000,B 90.000,C 0.000} C_DIS
LIN {X -79.937,Y -22.414,Z -20.773,A -90.000,B 90.000,C 0.000} C_DIS
LIN {X -79.797,Y -22.415,Z -20.756,A -90.000,B 90.000,C 0.000} C_DIS
LIN {X -79.610,Y -22.421,Z -20.742,A -90.000,B 90.000,C 0.000} C_DIS
LIN {X -79.479,Y -22.431,Z -20.741,A -90.000,B 90.000,C 0.000} C_DIS
LIN {X -79.330,Y -22.441,Z -20.746,A -90.000,B 90.000,C 0.000} C_DIS
LIN {X -79.091,Y -22.456,Z -20.755,A -90.000,B 90.000,C 0.000} C_DIS
LIN {X -78.717,Y -22.454,Z -20.782,A -90.000,B 90.000,C 0.000} C_DIS
LIN {X -78.574,Y -22.449,Z -20.800,A -90.000,B 90.000,C 0.000} C_DIS
LIN {X -78.409,Y -22.448,Z -20.828,A -90.000,B 90.000,C 0.000} C_DIS
LIN {X -78.159,Y -22.453,Z -20.885,A -90.000,B 90.000,C 0.000} C_DIS
LIN {X -78.006,Y -22.455,Z -20.922,A -90.000,B 90.000,C 0.000} C_DIS
LIN {X -77.894,Y -22.459,Z -20.954,A -90.000,B 90.000,C 0.000} C_DIS
LIN {X -77.825,Y -22.462,Z -20.978,A -90.000,B 90.000,C 0.000} C_DIS
LIN {X -77.724,Y -22.464,Z -21.019,A -90.000,B 90.000,C 0.000} C_DIS
LIN {X -77.508,Y -22.468,Z -21.113,A -90.000,B 90.000,C 0.000} C_DIS
LIN {X -77.473,Y -22.467,Z -21.129,A -90.000,B 90.000,C 0.000} C_DIS
LIN {X -77.186,Y -22.471,Z -21.288,A -90.000,B 90.000,C 0.000} C_DIS
LIN {X -76.793,Y -22.493,Z -21.544,A -90.000,B 90.000,C 0.000} C_DIS
LIN {X -76.614,Y -22.496,Z -21.665,A -90.000,B 90.000,C 0.000} C_DIS
LIN {X -76.457,Y -22.496,Z -21.776,A -90.000,B 90.000,C 0.000} C_DIS
LIN {X -76.343,Y -22.497,Z -21.865,A -90.000,B 90.000,C 0.000} C_DIS
LIN {X -76.245,Y -22.502,Z -21.952,A -90.000,B 90.000,C 0.000} C_DIS
LIN {X -76.030,Y -22.517,Z -22.152,A -90.000,B 90.000,C 0.000} C_DIS
LIN {X -75.900,Y -22.527,Z -22.289,A -90.000,B 90.000,C 0.000} C_DIS
LIN {X -75.820,Y -22.535,Z -22.382,A -90.000,B 90.000,C 0.000} C_DIS
LIN {X -75.431,Y -22.566,Z -22.841,A -90.000,B 90.000,C 0.000} C_DIS
LIN {X -75.137,Y -22.593,Z -23.200,A -90.000,B 90.000,C 0.000} C_DIS
LIN {X -75.036,Y -22.594,Z -23.296,A -90.000,B 90.000,C 0.000} C_DIS
LIN {X -74.788,Y -22.571,Z -23.453,A -90.000,B 90.000,C 0.000} C_DIS
LIN {X -74.617,Y -22.560,Z -23.552,A -90.000,B 90.000,C 0.000} C_DIS
LIN {X -74.490,Y -22.553,Z -23.631,A -90.000,B 90.000,C 0.000} C_DIS
LIN {X -74.051,Y -22.545,Z -23.925,A -90.000,B 90.000,C 0.000} C_DIS
LIN {X -73.824,Y -22.531,Z -24.080,A -90.000,B 90.000,C 0.000} C_DIS
LIN {X -73.575,Y -22.518,Z -24.256,A -90.000,B 90.000,C 0.000} C_DIS
LIN {X -73.318,Y -22.512,Z -24.442,A -90.000,B 90.000,C 0.000} C_DIS
LIN {X -73.165,Y -22.512,Z -24.565,A -90.000,B 90.000,C 0.000} C_DIS
LIN {X -72.933,Y -22.519,Z -24.784,A -90.000,B 90.000,C 0.000} C_DIS
LIN {X -72.586,Y -22.507,Z -25.145,A -90.000,B 90.000,C 0.000} C_DIS
LIN {X -72.083,Y -22.501,Z -25.667,A -90.000,B 90.000,C 0.000} C_DIS
LIN {X -71.981,Y -22.499,Z -25.781,A -90.000,B 90.000,C 0.000} C_DIS
LIN {X -71.902,Y -22.501,Z -25.884,A -90.000,B 90.000,C 0.000} C_DIS
LIN {X -71.730,Y -22.492,Z -26.131,A -90.000,B 90.000,C 0.000} C_DIS
LIN {X -71.669,Y -22.489,Z -26.227,A -90.000,B 90.000,C 0.000} C_DIS
LIN {X -71.571,Y -22.491,Z -26.411,A -90.000,B 90.000,C 0.000} C_DIS
LIN {X -71.420,Y -22.503,Z -26.716,A -90.000,B 90.000,C 0.000} C_DIS
LIN {X -71.281,Y -22.516,Z -27.008,A -90.000,B 90.000,C 0.000} C_DIS
LIN {X -71.183,Y -22.520,Z -27.218,A -90.000,B 90.000,C 0.000} C_DIS
LIN {X -71.129,Y -22.520,Z -27.321,A -90.000,B 90.000,C 0.000} C_DIS
LIN {X -71.061,Y -22.514,Z -27.455,A -90.000,B 90.000,C 0.000} C_DIS
LIN {X -71.007,Y -22.511,Z -27.571,A -90.000,B 90.000,C 0.000} C_DIS
LIN {X -70.920,Y -22.493,Z -27.771,A -90.000,B 90.000,C 0.000} C_DIS
LIN {X -70.890,Y -22.487,Z -27.846,A -90.000,B 90.000,C 0.000} C_DIS
LIN {X -70.855,Y -22.479,Z -27.950,A -90.000,B 90.000,C 0.000} C_DIS
LIN {X -70.838,Y -22.475,Z -28.005,A -90.000,B 90.000,C 0.000} C_DIS
LIN {X -70.750,Y -22.464,Z -28.342,A -90.000,B 90.000,C 0.000} C_DIS
LIN {X -70.726,Y -22.462,Z -28.447,A -90.000,B 90.000,C 0.000} C_DIS
LIN {X -70.659,Y -22.459,Z -28.781,A -90.000,B 90.000,C 0.000} C_DIS
LIN {X -70.642,Y -22.462,Z -28.899,A -90.000,B 90.000,C 0.000} C_DIS
LIN {X -70.602,Y -22.474,Z -29.227,A -90.000,B 90.000,C 0.000} C_DIS
LIN {X -70.595,Y -22.477,Z -29.298,A -90.000,B 90.000,C 0.000} C_DIS
LIN {X -70.573,Y -22.481,Z -29.580,A -90.000,B 90.000,C 0.000} C_DIS
LIN {X -70.552,Y -22.483,Z -29.895,A -90.000,B 90.000,C 0.000} C_DIS
LIN {X -70.539,Y -22.480,Z -30.131,A -90.000,B 90.000,C 0.000} C_DIS
LIN {X -70.537,Y -22.480,Z -30.219,A -90.000,B 90.000,C 0.000} C_DIS
LIN {X -70.537,Y -22.487,Z -30.633,A -90.000,B 90.000,C 0.000} C_DIS
LIN {X -70.538,Y -22.489,Z -30.715,A -90.000,B 90.000,C 0.000} C_DIS
LIN {X -70.554,Y -22.504,Z -31.170,A -90.000,B 90.000,C 0.000} C_DIS
LIN {X -70.557,Y -22.514,Z -31.311,A -90.000,B 90.000,C 0.000} C_DIS
LIN {X -70.585,Y -22.558,Z -32.222,A -90.000,B 90.000,C 0.000} C_DIS
LIN {X -70.601,Y -22.571,Z -32.395,A -90.000,B 90.000,C 0.000} C_DIS
LIN {X -70.638,Y -22.596,Z -32.665,A -90.000,B 90.000,C 0.000} C_DIS
LIN {X -70.642,Y -22.669,Z -33.094,A -90.000,B 90.000,C 0.000} C_DIS
LIN {X -70.631,Y -22.684,Z -33.212,A -90.000,B 90.000,C 0.000} C_DIS
LIN {X -70.621,Y -22.699,Z -33.327,A -90.000,B 90.000,C 0.000} C_DIS
LIN {X -70.574,Y -22.703,Z -33.449,A -90.000,B 90.000,C 0.000} C_DIS
LIN {X -70.367,Y -22.666,Z -33.656,A -90.000,B 90.000,C 0.000} C_DIS
LIN {X -70.041,Y -22.589,Z -33.879,A -90.000,B 90.000,C 0.000} C_DIS
LIN {X -69.747,Y -22.585,Z -34.053,A -90.000,B 90.000,C 0.000} C_DIS
LIN {X -69.655,Y -22.581,Z -34.102,A -90.000,B 90.000,C 0.000} C_DIS
LIN {X -69.317,Y -22.561,Z -34.258,A -90.000,B 90.000,C 0.000} C_DIS
LIN {X -69.162,Y -22.546,Z -34.332,A -90.000,B 90.000,C 0.000} C_DIS
LIN {X -69.023,Y -22.534,Z -34.403,A -90.000,B 90.000,C 0.000} C_DIS
LIN {X -67.860,Y -22.448,Z -35.020,A -90.000,B 90.000,C 0.000} C_DIS
LIN {X -67.610,Y -22.434,Z -35.163,A -90.000,B 90.000,C 0.000} C_DIS
LIN {X -66.810,Y -22.431,Z -35.595,A -90.000,B 90.000,C 0.000} C_DIS
LIN {X -66.412,Y -22.424,Z -35.796,A -90.000,B 90.000,C 0.000} C_DIS
LIN {X -65.264,Y -22.385,Z -36.385,A -90.000,B 90.000,C 0.000} C_DIS
LIN {X -64.877,Y -22.385,Z -36.577,A -90.000,B 90.000,C 0.000} C_DIS
LIN {X -64.383,Y -22.392,Z -36.837,A -90.000,B 90.000,C 0.000} C_DIS
LIN {X -63.572,Y -22.384,Z -37.223,A -90.000,B 90.000,C 0.000} C_DIS
LIN {X -62.696,Y -22.370,Z -37.643,A -90.000,B 90.000,C 0.000} C_DIS
LIN {X -62.137,Y -22.374,Z -37.903,A -90.000,B 90.000,C 0.000} C_DIS
LIN {X -61.855,Y -22.378,Z -38.040,A -90.000,B 90.000,C 0.000} C_DIS
LIN {X -60.889,Y -22.371,Z -38.461,A -90.000,B 90.000,C 0.000} C_DIS
LIN {X -60.069,Y -22.363,Z -38.821,A -90.000,B 90.000,C 0.000} C_DIS
LIN {X -59.480,Y -22.366,Z -39.075,A -90.000,B 90.000,C 0.000} C_DIS
LIN {X -59.249,Y -22.368,Z -39.173,A -90.000,B 90.000,C 0.000} C_DIS
LIN {X -57.604,Y -22.355,Z -39.807,A -90.000,B 90.000,C 0.000} C_DIS
LIN {X -56.804,Y -22.356,Z -40.111,A -90.000,B 90.000,C 0.000} C_DIS
LIN {X -56.229,Y -22.348,Z -40.304,A -90.000,B 90.000,C 0.000} C_DIS
LIN {X -54.997,Y -22.337,Z -40.721,A -90.000,B 90.000,C 0.000} C_DIS
LIN {X -54.089,Y -22.338,Z -41.022,A -90.000,B 90.000,C 0.000} C_DIS
LIN {X -53.570,Y -22.334,Z -41.185,A -90.000,B 90.000,C 0.000} C_DIS
LIN {X -52.062,Y -22.323,Z -41.631,A -90.000,B 90.000,C 0.000} C_DIS
LIN {X -51.309,Y -22.325,Z -41.849,A -90.000,B 90.000,C 0.000} C_DIS
LIN {X -50.164,Y -22.318,Z -42.162,A -90.000,B 90.000,C 0.000} C_DIS
LIN {X -49.548,Y -22.318,Z -42.328,A -90.000,B 90.000,C 0.000} C_DIS
LIN {X -48.549,Y -22.318,Z -42.583,A -90.000,B 90.000,C 0.000} C_DIS
LIN {X -47.992,Y -22.313,Z -42.709,A -90.000,B 90.000,C 0.000} C_DIS
LIN {X -47.039,Y -22.316,Z -42.937,A -90.000,B 90.000,C 0.000} C_DIS
LIN {X -45.995,Y -22.307,Z -43.172,A -90.000,B 90.000,C 0.000} C_DIS
LIN {X -45.577,Y -22.308,Z -43.279,A -90.000,B 90.000,C 0.000} C_DIS
LIN {X -44.332,Y -22.284,Z -43.550,A -90.000,B 90.000,C 0.000} C_DIS
LIN {X -43.952,Y -22.280,Z -43.638,A -90.000,B 90.000,C 0.000} C_DIS
LIN {X -43.100,Y -22.280,Z -43.852,A -90.000,B 90.000,C 0.000} C_DIS
LIN {X -42.473,Y -22.269,Z -44.016,A -90.000,B 90.000,C 0.000} C_DIS
LIN {X -41.942,Y -22.253,Z -44.144,A -90.000,B 90.000,C 0.000} C_DIS
LIN {X -41.754,Y -22.251,Z -44.194,A -90.000,B 90.000,C 0.000} C_DIS
LIN {X -41.199,Y -22.250,Z -44.338,A -90.000,B 90.000,C 0.000} C_DIS
LIN {X -41.018,Y -22.269,Z -44.372,A -90.000,B 90.000,C 0.000} C_DIS
LIN {X -40.510,Y -22.340,Z -44.461,A -90.000,B 90.000,C 0.000} C_DIS
LIN {X -39.929,Y -22.422,Z -44.567,A -90.000,B 90.000,C 0.000} C_DIS
LIN {X -39.445,Y -22.511,Z -44.650,A -90.000,B 90.000,C 0.000} C_DIS
LIN {X -39.112,Y -22.571,Z -44.710,A -90.000,B 90.000,C 0.000} C_DIS
LIN {X -39.018,Y -22.589,Z -44.730,A -90.000,B 90.000,C 0.000} C_DIS
LIN {X -38.537,Y -22.677,Z -44.842,A -90.000,B 90.000,C 0.000} C_DIS
LIN {X -38.340,Y -22.709,Z -44.889,A -90.000,B 90.000,C 0.000} C_DIS
LIN {X -37.986,Y -22.754,Z -44.978,A -90.000,B 90.000,C 0.000} C_DIS
LIN {X -37.314,Y -22.835,Z -45.152,A -90.000,B 90.000,C 0.000} C_DIS
LIN {X -36.269,Y -22.960,Z -45.428,A -90.000,B 90.000,C 0.000} C_DIS
LIN {X -35.847,Y -23.011,Z -45.544,A -90.000,B 90.000,C 0.000} C_DIS
LIN {X -35.201,Y -23.089,Z -45.749,A -90.000,B 90.000,C 0.000} C_DIS
LIN {X -34.771,Y -23.128,Z -45.889,A -90.000,B 90.000,C 0.000} C_DIS
LIN {X -34.754,Y -23.130,Z -45.798,A -90.000,B 90.000,C 0.000} C_DIS
LIN {X -34.703,Y -23.134,Z -45.552,A -90.000,B 90.000,C 0.000} C_DIS
LIN {X -34.667,Y -23.138,Z -45.419,A -90.000,B 90.000,C 0.000} C_DIS
LIN {X -34.641,Y -23.139,Z -45.339,A -90.000,B 90.000,C 0.000} C_DIS
LIN {X -34.593,Y -23.141,Z -45.217,A -90.000,B 90.000,C 0.000} C_DIS
LIN {X -34.552,Y -23.142,Z -45.129,A -90.000,B 90.000,C 0.000} C_DIS
LIN {X -34.493,Y -23.140,Z -45.019,A -90.000,B 90.000,C 0.000} C_DIS
LIN {X -34.419,Y -23.137,Z -44.900,A -90.000,B 90.000,C 0.000} C_DIS
LIN {X -34.338,Y -23.133,Z -44.779,A -90.000,B 90.000,C 0.000} C_DIS
LIN {X -34.217,Y -23.127,Z -44.618,A -90.000,B 90.000,C 0.000} C_DIS
LIN {X -34.185,Y -23.126,Z -44.580,A -90.000,B 90.000,C 0.000} C_DIS
LIN {X -34.129,Y -23.123,Z -44.518,A -90.000,B 90.000,C 0.000} C_DIS
LIN {X -33.974,Y -23.115,Z -44.361,A -90.000,B 90.000,C 0.000} C_DIS
LIN {X -33.905,Y -23.112,Z -44.295,A -90.000,B 90.000,C 0.000} C_DIS
LIN {X -33.751,Y -23.107,Z -44.167,A -90.000,B 90.000,C 0.000} C_DIS
LIN {X -33.117,Y -23.094,Z -43.694,A -90.000,B 90.000,C 0.000} C_DIS
LIN {X -33.009,Y -23.092,Z -43.618,A -90.000,B 90.000,C 0.000} C_DIS
LIN {X -32.895,Y -23.086,Z -43.549,A -90.000,B 90.000,C 0.000} C_DIS
LIN {X -32.470,Y -23.049,Z -43.296,A -90.000,B 90.000,C 0.000} C_DIS
LIN {X -31.909,Y -22.979,Z -42.968,A -90.000,B 90.000,C 0.000} C_DIS
LIN {X -31.752,Y -22.960,Z -42.883,A -90.000,B 90.000,C 0.000} C_DIS
LIN {X -31.438,Y -22.931,Z -42.745,A -90.000,B 90.000,C 0.000} C_DIS
LIN {X -31.382,Y -22.927,Z -42.726,A -90.000,B 90.000,C 0.000} C_DIS
LIN {X -31.199,Y -22.917,Z -42.678,A -90.000,B 90.000,C 0.000} C_DIS
LIN {X -31.028,Y -22.909,Z -42.639,A -90.000,B 90.000,C 0.000} C_DIS
LIN {X -30.661,Y -22.901,Z -42.595,A -90.000,B 90.000,C 0.000} C_DIS
LIN {X -30.559,Y -22.902,Z -42.595,A -90.000,B 90.000,C 0.000} C_DIS
LIN {X -29.147,Y -22.912,Z -42.612,A -90.000,B 90.000,C 0.000} C_DIS
LIN {X -28.760,Y -22.905,Z -42.622,A -90.000,B 90.000,C 0.000} C_DIS
LIN {X -28.409,Y -22.895,Z -42.615,A -90.000,B 90.000,C 0.000} C_DIS
LIN {X -27.804,Y -22.884,Z -42.606,A -90.000,B 90.000,C 0.000} C_DIS
LIN {X -27.023,Y -22.862,Z -42.598,A -90.000,B 90.000,C 0.000} C_DIS
LIN {X -26.472,Y -22.855,Z -42.622,A -90.000,B 90.000,C 0.000} C_DIS
LIN {X -26.110,Y -22.834,Z -42.577,A -90.000,B 90.000,C 0.000} C_DIS
LIN {X -26.022,Y -22.832,Z -42.566,A -90.000,B 90.000,C 0.000} C_DIS
LIN {X -25.823,Y -22.829,Z -42.549,A -90.000,B 90.000,C 0.000} C_DIS
LIN {X -24.973,Y -22.820,Z -42.485,A -90.000,B 90.000,C 0.000} C_DIS
LIN {X -24.835,Y -22.820,Z -42.479,A -90.000,B 90.000,C 0.000} C_DIS
LIN {X -24.552,Y -22.822,Z -42.477,A -90.000,B 90.000,C 0.000} C_DIS
LIN {X -24.336,Y -22.825,Z -42.482,A -90.000,B 90.000,C 0.000} C_DIS
LIN {X -24.087,Y -22.819,Z -42.458,A -90.000,B 90.000,C 0.000} C_DIS
LIN {X -23.305,Y -22.814,Z -42.419,A -90.000,B 90.000,C 0.000} C_DIS
LIN {X -22.393,Y -22.802,Z -42.378,A -90.000,B 90.000,C 0.000} C_DIS
LIN {X -21.860,Y -22.779,Z -42.302,A -90.000,B 90.000,C 0.000} C_DIS
LIN {X -20.579,Y -22.744,Z -42.115,A -90.000,B 90.000,C 0.000} C_DIS
LIN {X -20.350,Y -22.742,Z -42.095,A -90.000,B 90.000,C 0.000} C_DIS
LIN {X -19.956,Y -22.745,Z -42.081,A -90.000,B 90.000,C 0.000} C_DIS
LIN {X -19.422,Y -22.745,Z -42.056,A -90.000,B 90.000,C 0.000} C_DIS
LIN {X -18.979,Y -22.746,Z -42.040,A -90.000,B 90.000,C 0.000} C_DIS
LIN {X -17.276,Y -22.699,Z -41.997,A -90.000,B 90.000,C 0.000} C_DIS
LIN {X -16.388,Y -22.680,Z -41.995,A -90.000,B 90.000,C 0.000} C_DIS
LIN {X -16.378,Y -22.680,Z -41.995,A -90.000,B 90.000,C 0.000} C_DIS
LIN {X -15.540,Y -22.652,Z -41.994,A -90.000,B 90.000,C 0.000} C_DIS
LIN {X -14.820,Y -22.633,Z -41.992,A -90.000,B 90.000,C 0.000} C_DIS
LIN {X -14.433,Y -22.625,Z -41.999,A -90.000,B 90.000,C 0.000} C_DIS
LIN {X -14.101,Y -22.615,Z -42.007,A -90.000,B 90.000,C 0.000} C_DIS
LIN {X -13.994,Y -22.613,Z -42.012,A -90.000,B 90.000,C 0.000} C_DIS
LIN {X -13.240,Y -22.605,Z -42.068,A -90.000,B 90.000,C 0.000} C_DIS
LIN {X -12.932,Y -22.597,Z -42.092,A -90.000,B 90.000,C 0.000} C_DIS
LIN {X -12.847,Y -22.593,Z -42.102,A -90.000,B 90.000,C 0.000} C_DIS
LIN {X -11.165,Y -22.532,Z -42.322,A -90.000,B 90.000,C 0.000} C_DIS
LIN {X -10.504,Y -22.513,Z -42.411,A -90.000,B 90.000,C 0.000} C_DIS
LIN {X -9.935,Y -22.506,Z -42.506,A -90.000,B 90.000,C 0.000} C_DIS
LIN {X -9.057,Y -22.479,Z -42.659,A -90.000,B 90.000,C 0.000} C_DIS
LIN {X -7.731,Y -22.447,Z -42.914,A -90.000,B 90.000,C 0.000} C_DIS
LIN {X -7.157,Y -22.434,Z -43.026,A -90.000,B 90.000,C 0.000} C_DIS
LIN {X -6.752,Y -22.432,Z -43.119,A -90.000,B 90.000,C 0.000} C_DIS
LIN {X -6.441,Y -22.432,Z -43.196,A -90.000,B 90.000,C 0.000} C_DIS
LIN {X -6.238,Y -22.429,Z -43.251,A -90.000,B 90.000,C 0.000} C_DIS
LIN {X -5.310,Y -22.398,Z -43.509,A -90.000,B 90.000,C 0.000} C_DIS
LIN {X -3.964,Y -22.359,Z -43.891,A -90.000,B 90.000,C 0.000} C_DIS
LIN {X -3.801,Y -22.359,Z -43.943,A -90.000,B 90.000,C 0.000} C_DIS
LIN {X -3.455,Y -22.366,Z -44.068,A -90.000,B 90.000,C 0.000} C_DIS
LIN {X -1.816,Y -22.344,Z -44.696,A -90.000,B 90.000,C 0.000} C_DIS
LIN {X -1.656,Y -22.339,Z -44.754,A -90.000,B 90.000,C 0.000} C_DIS
LIN {X -1.307,Y -22.340,Z -44.897,A -90.000,B 90.000,C 0.000} C_DIS
LIN {X -1.078,Y -22.344,Z -44.996,A -90.000,B 90.000,C 0.000} C_DIS
LIN {X -0.458,Y -22.343,Z -45.285,A -90.000,B 90.000,C 0.000} C_DIS
LIN {X 0.286,Y -22.313,Z -45.584,A -90.000,B 90.000,C 0.000} C_DIS
LIN {X 0.623,Y -22.307,Z -45.731,A -90.000,B 90.000,C 0.000} C_DIS
LIN {X 0.844,Y -22.308,Z -45.836,A -90.000,B 90.000,C 0.000} C_DIS
LIN {X 1.981,Y -22.266,Z -46.318,A -90.000,B 90.000,C 0.000} C_DIS
LIN {X 2.606,Y -22.240,Z -46.576,A -90.000,B 90.000,C 0.000} C_DIS
LIN {X 3.014,Y -22.231,Z -46.739,A -90.000,B 90.000,C 0.000} C_DIS
LIN {X 3.198,Y -22.221,Z -46.804,A -90.000,B 90.000,C 0.000} C_DIS
LIN {X 3.791,Y -22.180,Z -46.999,A -90.000,B 90.000,C 0.000} C_DIS
LIN {X 3.923,Y -22.173,Z -47.046,A -90.000,B 90.000,C 0.000} C_DIS
LIN {X 4.334,Y -22.157,Z -47.194,A -90.000,B 90.000,C 0.000} C_DIS
LIN {X 4.694,Y -22.157,Z -47.314,A -90.000,B 90.000,C 0.000} C_DIS
LIN {X 5.770,Y -22.122,Z -47.624,A -90.000,B 90.000,C 0.000} C_DIS
LIN {X 5.881,Y -22.121,Z -47.658,A -90.000,B 90.000,C 0.000} C_DIS
LIN {X 5.980,Y -22.124,Z -47.686,A -90.000,B 90.000,C 0.000} C_DIS
LIN {X 6.211,Y -22.135,Z -47.749,A -90.000,B 90.000,C 0.000} C_DIS
LIN {X 6.372,Y -22.139,Z -47.787,A -90.000,B 90.000,C 0.000} C_DIS
LIN {X 6.526,Y -22.149,Z -47.819,A -90.000,B 90.000,C 0.000} C_DIS
LIN {X 7.019,Y -22.197,Z -47.910,A -90.000,B 90.000,C 0.000} C_DIS
LIN {X 7.158,Y -22.208,Z -47.939,A -90.000,B 90.000,C 0.000} C_DIS
LIN {X 7.441,Y -22.231,Z -48.008,A -90.000,B 90.000,C 0.000} C_DIS
LIN {X 7.691,Y -22.266,Z -48.060,A -90.000,B 90.000,C 0.000} C_DIS
LIN {X 7.801,Y -22.282,Z -48.082,A -90.000,B 90.000,C 0.000} C_DIS
LIN {X 8.499,Y -22.384,Z -48.200,A -90.000,B 90.000,C 0.000} C_DIS
LIN {X 8.704,Y -22.417,Z -48.235,A -90.000,B 90.000,C 0.000} C_DIS
LIN {X 9.171,Y -22.495,Z -48.326,A -90.000,B 90.000,C 0.000} C_DIS
LIN {X 9.615,Y -22.573,Z -48.428,A -90.000,B 90.000,C 0.000} C_DIS
LIN {X 9.817,Y -22.614,Z -48.473,A -90.000,B 90.000,C 0.000} C_DIS
LIN {X 10.232,Y -22.695,Z -48.556,A -90.000,B 90.000,C 0.000} C_DIS
LIN {X 10.686,Y -22.785,Z -48.651,A -90.000,B 90.000,C 0.000} C_DIS
LIN {X 10.931,Y -22.760,Z -48.281,A -90.000,B 90.000,C 0.000} C_DIS
LIN {X 10.979,Y -22.755,Z -48.212,A -90.000,B 90.000,C 0.000} C_DIS
LIN {X 11.066,Y -22.745,Z -48.103,A -90.000,B 90.000,C 0.000} C_DIS
LIN {X 11.168,Y -22.737,Z -47.991,A -90.000,B 90.000,C 0.000} C_DIS
LIN {X 11.358,Y -22.724,Z -47.793,A -90.000,B 90.000,C 0.000} C_DIS
LIN {X 11.499,Y -22.716,Z -47.664,A -90.000,B 90.000,C 0.000} C_DIS
LIN {X 11.593,Y -22.713,Z -47.589,A -90.000,B 90.000,C 0.000} C_DIS
LIN {X 11.824,Y -22.709,Z -47.417,A -90.000,B 90.000,C 0.000} C_DIS
LIN {X 12.026,Y -22.689,Z -47.210,A -90.000,B 90.000,C 0.000} C_DIS
LIN {X 12.078,Y -22.685,Z -47.160,A -90.000,B 90.000,C 0.000} C_DIS
LIN {X 12.201,Y -22.681,Z -47.052,A -90.000,B 90.000,C 0.000} C_DIS
LIN {X 12.261,Y -22.678,Z -47.007,A -90.000,B 90.000,C 0.000} C_DIS
LIN {X 12.465,Y -22.663,Z -46.859,A -90.000,B 90.000,C 0.000} C_DIS
LIN {X 12.558,Y -22.655,Z -46.796,A -90.000,B 90.000,C 0.000} C_DIS
LIN {X 12.703,Y -22.645,Z -46.704,A -90.000,B 90.000,C 0.000} C_DIS
LIN {X 13.133,Y -22.613,Z -46.430,A -90.000,B 90.000,C 0.000} C_DIS
LIN {X 13.361,Y -22.586,Z -46.263,A -90.000,B 90.000,C 0.000} C_DIS
LIN {X 13.395,Y -22.582,Z -46.238,A -90.000,B 90.000,C 0.000} C_DIS
LIN {X 13.580,Y -22.565,Z -46.122,A -90.000,B 90.000,C 0.000} C_DIS
LIN {X 13.676,Y -22.559,Z -46.068,A -90.000,B 90.000,C 0.000} C_DIS
LIN {X 13.827,Y -22.540,Z -45.986,A -90.000,B 90.000,C 0.000} C_DIS
LIN {X 13.930,Y -22.529,Z -45.934,A -90.000,B 90.000,C 0.000} C_DIS
LIN {X 14.047,Y -22.518,Z -45.878,A -90.000,B 90.000,C 0.000} C_DIS
LIN {X 14.318,Y -22.481,Z -45.724,A -90.000,B 90.000,C 0.000} C_DIS
LIN {X 14.685,Y -22.425,Z -45.533,A -90.000,B 90.000,C 0.000} C_DIS
LIN {X 14.900,Y -22.400,Z -45.436,A -90.000,B 90.000,C 0.000} C_DIS
LIN {X 15.017,Y -22.393,Z -45.392,A -90.000,B 90.000,C 0.000} C_DIS
LIN {X 15.293,Y -22.369,Z -45.295,A -90.000,B 90.000,C 0.000} C_DIS
LIN {X 16.277,Y -22.292,Z -45.000,A -90.000,B 90.000,C 0.000} C_DIS
LIN {X 16.458,Y -22.268,Z -44.931,A -90.000,B 90.000,C 0.000} C_DIS
LIN {X 16.594,Y -22.253,Z -44.887,A -90.000,B 90.000,C 0.000} C_DIS
LIN {X 16.942,Y -22.220,Z -44.783,A -90.000,B 90.000,C 0.000} C_DIS
LIN {X 17.564,Y -22.160,Z -44.643,A -90.000,B 90.000,C 0.000} C_DIS
LIN {X 17.848,Y -22.136,Z -44.585,A -90.000,B 90.000,C 0.000} C_DIS
LIN {X 17.906,Y -22.130,Z -44.571,A -90.000,B 90.000,C 0.000} C_DIS
LIN {X 18.186,Y -22.112,Z -44.503,A -90.000,B 90.000,C 0.000} C_DIS
LIN {X 18.795,Y -22.067,Z -44.380,A -90.000,B 90.000,C 0.000} C_DIS
LIN {X 19.033,Y -22.053,Z -44.339,A -90.000,B 90.000,C 0.000} C_DIS
LIN {X 19.274,Y -22.038,Z -44.302,A -90.000,B 90.000,C 0.000} C_DIS
LIN {X 19.346,Y -22.035,Z -44.292,A -90.000,B 90.000,C 0.000} C_DIS
LIN {X 19.904,Y -21.987,Z -44.189,A -90.000,B 90.000,C 0.000} C_DIS
LIN {X 20.475,Y -21.932,Z -44.099,A -90.000,B 90.000,C 0.000} C_DIS
LIN {X 20.759,Y -21.915,Z -44.050,A -90.000,B 90.000,C 0.000} C_DIS
LIN {X 20.927,Y -21.903,Z -44.022,A -90.000,B 90.000,C 0.000} C_DIS
LIN {X 21.031,Y -21.898,Z -44.006,A -90.000,B 90.000,C 0.000} C_DIS
LIN {X 21.170,Y -21.894,Z -43.989,A -90.000,B 90.000,C 0.000} C_DIS
LIN {X 21.700,Y -21.874,Z -43.925,A -90.000,B 90.000,C 0.000} C_DIS
LIN {X 22.085,Y -21.839,Z -43.861,A -90.000,B 90.000,C 0.000} C_DIS
LIN {X 22.664,Y -21.791,Z -43.768,A -90.000,B 90.000,C 0.000} C_DIS
LIN {X 22.887,Y -21.782,Z -43.740,A -90.000,B 90.000,C 0.000} C_DIS
LIN {X 23.379,Y -21.774,Z -43.665,A -90.000,B 90.000,C 0.000} C_DIS
LIN {X 23.648,Y -21.767,Z -43.626,A -90.000,B 90.000,C 0.000} C_DIS
LIN {X 24.041,Y -21.739,Z -43.553,A -90.000,B 90.000,C 0.000} C_DIS
LIN {X 24.157,Y -21.734,Z -43.534,A -90.000,B 90.000,C 0.000} C_DIS
LIN {X 24.855,Y -21.716,Z -43.427,A -90.000,B 90.000,C 0.000} C_DIS
LIN {X 25.310,Y -21.712,Z -43.338,A -90.000,B 90.000,C 0.000} C_DIS
LIN {X 25.742,Y -21.713,Z -43.255,A -90.000,B 90.000,C 0.000} C_DIS
LIN {X 25.928,Y -21.710,Z -43.215,A -90.000,B 90.000,C 0.000} C_DIS
LIN {X 26.034,Y -21.709,Z -43.193,A -90.000,B 90.000,C 0.000} C_DIS
LIN {X 26.473,Y -21.705,Z -43.100,A -90.000,B 90.000,C 0.000} C_DIS
LIN {X 26.959,Y -21.705,Z -42.995,A -90.000,B 90.000,C 0.000} C_DIS
LIN {X 27.316,Y -21.719,Z -42.914,A -90.000,B 90.000,C 0.000} C_DIS
LIN {X 27.534,Y -21.729,Z -42.863,A -90.000,B 90.000,C 0.000} C_DIS
LIN {X 27.745,Y -21.734,Z -42.809,A -90.000,B 90.000,C 0.000} C_DIS
LIN {X 28.472,Y -21.742,Z -42.613,A -90.000,B 90.000,C 0.000} C_DIS
LIN {X 28.802,Y -21.748,Z -42.526,A -90.000,B 90.000,C 0.000} C_DIS
LIN {X 28.946,Y -21.748,Z -42.484,A -90.000,B 90.000,C 0.000} C_DIS
LIN {X 29.843,Y -21.762,Z -42.206,A -90.000,B 90.000,C 0.000} C_DIS
LIN {X 30.207,Y -21.761,Z -42.089,A -90.000,B 90.000,C 0.000} C_DIS
LIN {X 30.965,Y -21.749,Z -41.839,A -90.000,B 90.000,C 0.000} C_DIS
LIN {X 31.332,Y -21.738,Z -41.725,A -90.000,B 90.000,C 0.000} C_DIS
LIN {X 32.438,Y -21.728,Z -41.354,A -90.000,B 90.000,C 0.000} C_DIS
LIN {X 32.834,Y -21.721,Z -41.226,A -90.000,B 90.000,C 0.000} C_DIS
LIN {X 33.995,Y -21.688,Z -40.858,A -90.000,B 90.000,C 0.000} C_DIS
LIN {X 34.154,Y -21.682,Z -40.809,A -90.000,B 90.000,C 0.000} C_DIS
LIN {X 34.437,Y -21.668,Z -40.736,A -90.000,B 90.000,C 0.000} C_DIS
LIN {X 35.294,Y -21.645,Z -40.500,A -90.000,B 90.000,C 0.000} C_DIS
LIN {X 35.509,Y -21.640,Z -40.442,A -90.000,B 90.000,C 0.000} C_DIS
LIN {X 36.077,Y -21.629,Z -40.302,A -90.000,B 90.000,C 0.000} C_DIS
LIN {X 36.905,Y -21.596,Z -40.122,A -90.000,B 90.000,C 0.000} C_DIS
LIN {X 37.482,Y -21.587,Z -40.005,A -90.000,B 90.000,C 0.000} C_DIS
LIN {X 38.094,Y -21.560,Z -39.913,A -90.000,B 90.000,C 0.000} C_DIS
LIN {X 38.382,Y -21.550,Z -39.873,A -90.000,B 90.000,C 0.000} C_DIS
LIN {X 38.945,Y -21.528,Z -39.803,A -90.000,B 90.000,C 0.000} C_DIS
LIN {X 39.439,Y -21.523,Z -39.749,A -90.000,B 90.000,C 0.000} C_DIS
LIN {X 39.897,Y -21.515,Z -39.705,A -90.000,B 90.000,C 0.000} C_DIS
LIN {X 40.652,Y -21.484,Z -39.676,A -90.000,B 90.000,C 0.000} C_DIS
LIN {X 40.899,Y -21.475,Z -39.667,A -90.000,B 90.000,C 0.000} C_DIS
LIN {X 41.186,Y -21.470,Z -39.659,A -90.000,B 90.000,C 0.000} C_DIS
LIN {X 41.451,Y -21.463,Z -39.657,A -90.000,B 90.000,C 0.000} C_DIS
LIN {X 41.894,Y -21.455,Z -39.663,A -90.000,B 90.000,C 0.000} C_DIS
LIN {X 42.360,Y -21.443,Z -39.681,A -90.000,B 90.000,C 0.000} C_DIS
LIN {X 43.069,Y -21.424,Z -39.734,A -90.000,B 90.000,C 0.000} C_DIS
LIN {X 43.548,Y -21.411,Z -39.783,A -90.000,B 90.000,C 0.000} C_DIS
LIN {X 43.950,Y -21.404,Z -39.825,A -90.000,B 90.000,C 0.000} C_DIS
LIN {X 44.338,Y -21.400,Z -39.873,A -90.000,B 90.000,C 0.000} C_DIS
LIN {X 44.402,Y -21.400,Z -39.881,A -90.000,B 90.000,C 0.000} C_DIS
LIN {X 44.873,Y -21.395,Z -39.962,A -90.000,B 90.000,C 0.000} C_DIS
LIN {X 45.193,Y -21.391,Z -40.021,A -90.000,B 90.000,C 0.000} C_DIS
LIN {X 45.941,Y -21.371,Z -40.206,A -90.000,B 90.000,C 0.000} C_DIS
LIN {X 46.411,Y -21.367,Z -40.325,A -90.000,B 90.000,C 0.000} C_DIS
LIN {X 46.871,Y -21.361,Z -40.454,A -90.000,B 90.000,C 0.000} C_DIS
LIN {X 47.892,Y -21.344,Z -40.773,A -90.000,B 90.000,C 0.000} C_DIS
LIN {X 48.282,Y -21.341,Z -40.895,A -90.000,B 90.000,C 0.000} C_DIS
LIN {X 48.625,Y -21.343,Z -41.005,A -90.000,B 90.000,C 0.000} C_DIS
LIN {X 49.074,Y -21.343,Z -41.185,A -90.000,B 90.000,C 0.000} C_DIS
LIN {X 49.982,Y -21.336,Z -41.584,A -90.000,B 90.000,C 0.000} C_DIS
LIN {X 50.472,Y -21.331,Z -41.817,A -90.000,B 90.000,C 0.000} C_DIS
LIN {X 51.125,Y -21.327,Z -42.128,A -90.000,B 90.000,C 0.000} C_DIS
LIN {X 51.579,Y -21.324,Z -42.351,A -90.000,B 90.000,C 0.000} C_DIS
LIN {X 51.850,Y -21.325,Z -42.485,A -90.000,B 90.000,C 0.000} C_DIS
LIN {X 52.293,Y -21.325,Z -42.723,A -90.000,B 90.000,C 0.000} C_DIS
LIN {X 54.617,Y -21.316,Z -44.108,A -90.000,B 90.000,C 0.000} C_DIS
LIN {X 54.892,Y -21.317,Z -44.273,A -90.000,B 90.000,C 0.000} C_DIS
LIN {X 55.296,Y -21.318,Z -44.546,A -90.000,B 90.000,C 0.000} C_DIS
LIN {X 55.346,Y -21.318,Z -44.582,A -90.000,B 90.000,C 0.000} C_DIS
LIN {X 56.512,Y -21.317,Z -45.441,A -90.000,B 90.000,C 0.000} C_DIS
LIN {X 57.250,Y -21.315,Z -45.995,A -90.000,B 90.000,C 0.000} C_DIS
LIN {X 57.589,Y -21.316,Z -46.239,A -90.000,B 90.000,C 0.000} C_DIS
LIN {X 57.962,Y -21.316,Z -46.554,A -90.000,B 90.000,C 0.000} C_DIS
LIN {X 59.526,Y -21.315,Z -47.894,A -90.000,B 90.000,C 0.000} C_DIS
LIN {X 60.025,Y -21.315,Z -48.330,A -90.000,B 90.000,C 0.000} C_DIS
LIN {X 61.908,Y -21.318,Z -50.068,A -90.000,B 90.000,C 0.000} C_DIS
LIN {X 62.459,Y -21.321,Z -50.545,A -90.000,B 90.000,C 0.000} C_DIS
LIN {X 63.558,Y -21.324,Z -51.542,A -90.000,B 90.000,C 0.000} C_DIS
LIN {X 63.753,Y -21.327,Z -51.693,A -90.000,B 90.000,C 0.000} C_DIS
LIN {X 64.761,Y -21.333,Z -52.478,A -90.000,B 90.000,C 0.000} C_DIS
LIN {X 65.200,Y -21.334,Z -52.832,A -90.000,B 90.000,C 0.000} C_DIS
LIN {X 65.422,Y -21.340,Z -52.977,A -90.000,B 90.000,C 0.000} C_DIS
LIN {X 66.456,Y -21.344,Z -53.649,A -90.000,B 90.000,C 0.000} C_DIS
LIN {X 67.074,Y -21.350,Z -54.028,A -90.000,B 90.000,C 0.000} C_DIS
LIN {X 68.350,Y -21.354,Z -54.789,A -90.000,B 90.000,C 0.000} C_DIS
LIN {X 69.159,Y -21.358,Z -55.260,A -90.000,B 90.000,C 0.000} C_DIS
LIN {X 70.395,Y -21.361,Z -56.005,A -90.000,B 90.000,C 0.000} C_DIS
LIN {X 71.295,Y -21.364,Z -56.542,A -90.000,B 90.000,C 0.000} C_DIS
LIN {X 71.787,Y -21.364,Z -56.870,A -90.000,B 90.000,C 0.000} C_DIS
LIN {X 72.570,Y -21.366,Z -57.395,A -90.000,B 90.000,C 0.000} C_DIS
LIN {X 73.658,Y -21.370,Z -58.118,A -90.000,B 90.000,C 0.000} C_DIS
LIN {X 74.619,Y -21.373,Z -58.897,A -90.000,B 90.000,C 0.000} C_DIS
LIN {X 75.657,Y -21.381,Z -59.759,A -90.000,B 90.000,C 0.000} C_DIS
LIN {X 76.366,Y -21.385,Z -60.445,A -90.000,B 90.000,C 0.000} C_DIS
LIN {X 76.945,Y -21.396,Z -61.010,A -90.000,B 90.000,C 0.000} C_DIS
LIN {X 77.346,Y -21.401,Z -61.413,A -90.000,B 90.000,C 0.000} C_DIS
LIN {X 77.413,Y -21.402,Z -61.482,A -90.000,B 90.000,C 0.000} C_DIS
LIN {X 77.655,Y -21.405,Z -61.754,A -90.000,B 90.000,C 0.000} C_DIS
LIN {X 78.334,Y -21.423,Z -62.525,A -90.000,B 90.000,C 0.000} C_DIS
LIN {X 78.600,Y -21.427,Z -62.845,A -90.000,B 90.000,C 0.000} C_DIS
LIN {X 78.674,Y -21.395,Z -62.919,A -90.000,B 90.000,C 0.000} C_DIS
LIN {X 78.921,Y -21.326,Z -63.184,A -90.000,B 90.000,C 0.000} C_DIS
LIN {X 78.980,Y -21.317,Z -63.254,A -90.000,B 90.000,C 0.000} C_DIS
LIN {X 79.062,Y -21.310,Z -63.353,A -90.000,B 90.000,C 0.000} C_DIS
LIN {X 79.119,Y -21.308,Z -63.424,A -90.000,B 90.000,C 0.000} C_DIS
LIN {X 79.119,Y -60.000,Z -63.424,A -90.000,B 90.000,C 0.000} C_DIS
LIN {X 105.409,Y -60.000,Z -76.519,A -90.000,B 90.000,C 0.000} C_DIS
LIN {X 105.409,Y -21.308,Z -76.519,A -90.000,B 90.000,C 0.000} C_DIS
LIN {X 105.346,Y -21.308,Z -76.638,A -90.000,B 90.000,C 0.000} C_DIS
LIN {X 105.346,Y -60.000,Z -76.638,A -90.000,B 90.000,C 0.000} C_DIS
LIN {X 99.856,Y -60.000,Z -87.283,A -90.000,B 90.000,C 0.000} C_DIS
LIN {X 99.856,Y -21.308,Z -87.283,A -90.000,B 90.000,C 0.000} C_DIS
LIN {X 99.858,Y -21.308,Z -87.310,A -90.000,B 90.000,C 0.000} C_DIS
LIN {X 99.876,Y -24.476,Z -87.534,A -90.000,B 90.000,C 0.000} C_DIS
LIN {X 99.878,Y -24.474,Z -87.562,A -90.000,B 90.000,C 0.000} C_DIS
LIN {X 99.878,Y -24.485,Z -87.566,A -90.000,B 90.000,C 0.000} C_DIS
LIN {X 99.878,Y -24.530,Z -87.570,A -90.000,B 90.000,C 0.000} C_DIS
LIN {X 99.879,Y -24.568,Z -87.598,A -90.000,B 90.000,C 0.000} C_DIS
LIN {X 99.894,Y -21.308,Z -87.822,A -90.000,B 90.000,C 0.000} C_DIS
LIN {X 99.985,Y -21.329,Z -89.106,A -90.000,B 90.000,C 0.000} C_DIS
LIN {X 100.002,Y -21.308,Z -89.349,A -90.000,B 90.000,C 0.000} C_DIS
LIN {X 100.002,Y -60.000,Z -89.349,A -90.000,B 90.000,C 0.000} C_DIS
LIN {X 117.211,Y -60.000,Z -45.905,A -90.000,B 90.000,C 0.000} C_DIS
LIN {X 117.211,Y -21.308,Z -45.905,A -90.000,B 90.000,C 0.000} C_DIS
LIN {X 117.204,Y -21.308,Z -45.929,A -90.000,B 90.000,C 0.000} C_DIS
LIN {X 117.158,Y -36.147,Z -46.078,A -90.000,B 90.000,C 0.000} C_DIS
LIN {X 117.113,Y -36.161,Z -46.218,A -90.000,B 90.000,C 0.000} C_DIS
LIN {X 117.079,Y -36.191,Z -46.317,A -90.000,B 90.000,C 0.000} C_DIS
LIN {X 117.024,Y -36.262,Z -46.469,A -90.000,B 90.000,C 0.000} C_DIS
LIN {X 116.979,Y -36.330,Z -46.582,A -90.000,B 90.000,C 0.000} C_DIS
LIN {X 116.936,Y -36.402,Z -46.685,A -90.000,B 90.000,C 0.000} C_DIS
LIN {X 116.892,Y -36.478,Z -46.779,A -90.000,B 90.000,C 0.000} C_DIS
LIN {X 116.849,Y -36.557,Z -46.865,A -90.000,B 90.000,C 0.000} C_DIS
LIN {X 116.806,Y -36.639,Z -46.943,A -90.000,B 90.000,C 0.000} C_DIS
LIN {X 116.764,Y -36.727,Z -47.012,A -90.000,B 90.000,C 0.000} C_DIS
LIN {X 116.743,Y -36.774,Z -47.044,A -90.000,B 90.000,C 0.000} C_DIS
LIN {X 116.701,Y -36.873,Z -47.101,A -90.000,B 90.000,C 0.000} C_DIS
LIN {X 116.640,Y -37.027,Z -47.173,A -90.000,B 90.000,C 0.000} C_DIS
LIN {X 116.579,Y -37.178,Z -47.227,A -90.000,B 90.000,C 0.000} C_DIS
LIN {X 116.519,Y -37.329,Z -47.264,A -90.000,B 90.000,C 0.000} C_DIS
LIN {X 116.479,Y -37.433,Z -47.280,A -90.000,B 90.000,C 0.000} C_DIS
LIN {X 116.460,Y -37.486,Z -47.285,A -90.000,B 90.000,C 0.000} C_DIS
LIN {X 116.421,Y -37.600,Z -47.290,A -90.000,B 90.000,C 0.000} C_DIS
LIN {X 116.364,Y -37.781,Z -47.285,A -90.000,B 90.000,C 0.000} C_DIS
LIN {X 116.308,Y -37.959,Z -47.266,A -90.000,B 90.000,C 0.000} C_DIS
LIN {X 116.271,Y -38.079,Z -47.244,A -90.000,B 90.000,C 0.000} C_DIS
LIN {X 116.235,Y -38.205,Z -47.217,A -90.000,B 90.000,C 0.000} C_DIS
LIN {X 116.199,Y -38.337,Z -47.183,A -90.000,B 90.000,C 0.000} C_DIS
LIN {X 116.147,Y -38.550,Z -47.122,A -90.000,B 90.000,C 0.000} C_DIS
LIN {X 116.112,Y -38.684,Z -47.074,A -90.000,B 90.000,C 0.000} C_DIS
LIN {X 116.045,Y -38.956,Z -46.961,A -90.000,B 90.000,C 0.000} C_DIS
LIN {X 116.013,Y -39.090,Z -46.897,A -90.000,B 90.000,C 0.000} C_DIS
LIN {X 115.980,Y -39.216,Z -46.827,A -90.000,B 90.000,C 0.000} C_DIS
LIN {X 115.949,Y -39.335,Z -46.753,A -90.000,B 90.000,C 0.000} C_DIS
LIN {X 115.888,Y -39.572,Z -46.590,A -90.000,B 90.000,C 0.000} C_DIS
LIN {X 115.858,Y -39.688,Z -46.501,A -90.000,B 90.000,C 0.000} C_DIS
LIN {X 115.829,Y -39.796,Z -46.408,A -90.000,B 90.000,C 0.000} C_DIS
LIN {X 115.800,Y -39.896,Z -46.311,A -90.000,B 90.000,C 0.000} C_DIS
LIN {X 115.772,Y -39.991,Z -46.210,A -90.000,B 90.000,C 0.000} C_DIS
LIN {X 115.718,Y -40.173,Z -45.996,A -90.000,B 90.000,C 0.000} C_DIS
LIN {X 115.692,Y -40.265,Z -45.884,A -90.000,B 90.000,C 0.000} C_DIS
LIN {X 115.667,Y -40.352,Z -45.768,A -90.000,B 90.000,C 0.000} C_DIS
LIN {X 115.643,Y -40.435,Z -45.648,A -90.000,B 90.000,C 0.000} C_DIS
LIN {X 115.619,Y -40.513,Z -45.526,A -90.000,B 90.000,C 0.000} C_DIS
LIN {X 115.596,Y -40.586,Z -45.400,A -90.000,B 90.000,C 0.000} C_DIS
LIN {X 115.530,Y -40.805,Z -45.007,A -90.000,B 90.000,C 0.000} C_DIS
LIN {X 115.510,Y -40.876,Z -44.870,A -90.000,B 90.000,C 0.000} C_DIS
LIN {X 115.490,Y -40.962,Z -44.732,A -90.000,B 90.000,C 0.000} C_DIS
LIN {X 115.472,Y -41.064,Z -44.591,A -90.000,B 90.000,C 0.000} C_DIS
LIN {X 115.454,Y -41.171,Z -44.448,A -90.000,B 90.000,C 0.000} C_DIS
LIN {X 115.420,Y -41.359,Z -44.158,A -90.000,B 90.000,C 0.000} C_DIS
LIN {X 115.389,Y -41.530,Z -43.861,A -90.000,B 90.000,C 0.000} C_DIS
LIN {X 115.362,Y -41.672,Z -43.559,A -90.000,B 90.000,C 0.000} C_DIS
LIN {X 115.338,Y -41.780,Z -43.253,A -90.000,B 90.000,C 0.000} C_DIS
LIN {X 115.317,Y -41.867,Z -42.945,A -90.000,B 90.000,C 0.000} C_DIS
LIN {X 115.300,Y -41.930,Z -42.635,A -90.000,B 90.000,C 0.000} C_DIS
LIN {X 115.286,Y -41.961,Z -42.325,A -90.000,B 90.000,C 0.000} C_DIS
LIN {X 115.276,Y -41.971,Z -42.015,A -90.000,B 90.000,C 0.000} C_DIS
LIN {X 115.269,Y -41.959,Z -41.708,A -90.000,B 90.000,C 0.000} C_DIS
LIN {X 115.266,Y -41.923,Z -41.405,A -90.000,B 90.000,C 0.000} C_DIS
LIN {X 115.267,Y -41.871,Z -41.106,A -90.000,B 90.000,C 0.000} C_DIS
LIN {X 115.269,Y -41.836,Z -40.958,A -90.000,B 90.000,C 0.000} C_DIS
LIN {X 115.272,Y -41.796,Z -40.812,A -90.000,B 90.000,C 0.000} C_DIS
LIN {X 115.281,Y -41.707,Z -40.525,A -90.000,B 90.000,C 0.000} C_DIS
LIN {X 115.286,Y -41.656,Z -40.385,A -90.000,B 90.000,C 0.000} C_DIS
LIN {X 115.293,Y -41.598,Z -40.247,A -90.000,B 90.000,C 0.000} C_DIS
LIN {X 115.301,Y -41.533,Z -40.111,A -90.000,B 90.000,C 0.000} C_DIS
LIN {X 115.310,Y -41.462,Z -39.978,A -90.000,B 90.000,C 0.000} C_DIS
LIN {X 115.320,Y -41.387,Z -39.847,A -90.000,B 90.000,C 0.000} C_DIS
LIN {X 115.331,Y -41.308,Z -39.719,A -90.000,B 90.000,C 0.000} C_DIS
LIN {X 115.343,Y -41.224,Z -39.594,A -90.000,B 90.000,C 0.000} C_DIS
LIN {X 115.356,Y -41.135,Z -39.472,A -90.000,B 90.000,C 0.000} C_DIS
LIN {X 115.371,Y -41.043,Z -39.353,A -90.000,B 90.000,C 0.000} C_DIS
LIN {X 115.386,Y -40.947,Z -39.238,A -90.000,B 90.000,C 0.000} C_DIS
LIN {X 115.402,Y -40.847,Z -39.126,A -90.000,B 90.000,C 0.000} C_DIS
LIN {X 115.420,Y -40.739,Z -39.018,A -90.000,B 90.000,C 0.000} C_DIS
LIN {X 115.438,Y -40.625,Z -38.913,A -90.000,B 90.000,C 0.000} C_DIS
LIN {X 115.458,Y -40.503,Z -38.813,A -90.000,B 90.000,C 0.000} C_DIS
LIN {X 115.479,Y -40.373,Z -38.717,A -90.000,B 90.000,C 0.000} C_DIS
LIN {X 115.501,Y -40.239,Z -38.624,A -90.000,B 90.000,C 0.000} C_DIS
LIN {X 115.524,Y -40.108,Z -38.537,A -90.000,B 90.000,C 0.000} C_DIS
LIN {X 115.548,Y -39.976,Z -38.454,A -90.000,B 90.000,C 0.000} C_DIS
LIN {X 115.573,Y -39.839,Z -38.375,A -90.000,B 90.000,C 0.000} C_DIS
LIN {X 115.600,Y -39.708,Z -38.302,A -90.000,B 90.000,C 0.000} C_DIS
LIN {X 115.628,Y -39.575,Z -38.233,A -90.000,B 90.000,C 0.000} C_DIS
LIN {X 115.657,Y -39.442,Z -38.170,A -90.000,B 90.000,C 0.000} C_DIS
LIN {X 115.687,Y -39.313,Z -38.111,A -90.000,B 90.000,C 0.000} C_DIS
LIN {X 115.734,Y -39.114,Z -38.035,A -90.000,B 90.000,C 0.000} C_DIS
LIN {X 115.785,Y -38.910,Z -37.970,A -90.000,B 90.000,C 0.000} C_DIS
LIN {X 115.838,Y -38.717,Z -37.919,A -90.000,B 90.000,C 0.000} C_DIS
LIN {X 115.893,Y -38.518,Z -37.882,A -90.000,B 90.000,C 0.000} C_DIS
LIN {X 115.932,Y -38.379,Z -37.865,A -90.000,B 90.000,C 0.000} C_DIS
LIN {X 115.993,Y -38.161,Z -37.852,A -90.000,B 90.000,C 0.000} C_DIS
LIN {X 116.035,Y -38.030,Z -37.852,A -90.000,B 90.000,C 0.000} C_DIS
LIN {X 116.100,Y -37.846,Z -37.864,A -90.000,B 90.000,C 0.000} C_DIS
LIN {X 116.145,Y -37.727,Z -37.881,A -90.000,B 90.000,C 0.000} C_DIS
LIN {X 116.192,Y -37.615,Z -37.906,A -90.000,B 90.000,C 0.000} C_DIS
LIN {X 116.240,Y -37.506,Z -37.937,A -90.000,B 90.000,C 0.000} C_DIS
LIN {X 116.289,Y -37.401,Z -37.977,A -90.000,B 90.000,C 0.000} C_DIS
LIN {X 116.339,Y -37.305,Z -38.023,A -90.000,B 90.000,C 0.000} C_DIS
LIN {X 116.391,Y -37.223,Z -38.078,A -90.000,B 90.000,C 0.000} C_DIS
LIN {X 116.444,Y -37.153,Z -38.141,A -90.000,B 90.000,C 0.000} C_DIS
LIN {X 116.499,Y -37.097,Z -38.212,A -90.000,B 90.000,C 0.000} C_DIS
LIN {X 116.555,Y -37.054,Z -38.291,A -90.000,B 90.000,C 0.000} C_DIS
LIN {X 116.612,Y -37.025,Z -38.378,A -90.000,B 90.000,C 0.000} C_DIS
LIN {X 116.671,Y -37.009,Z -38.475,A -90.000,B 90.000,C 0.000} C_DIS
LIN {X 116.731,Y -37.005,Z -38.579,A -90.000,B 90.000,C 0.000} C_DIS
LIN {X 116.793,Y -37.011,Z -38.693,A -90.000,B 90.000,C 0.000} C_DIS
LIN {X 116.856,Y -37.001,Z -38.816,A -90.000,B 90.000,C 0.000} C_DIS
LIN {X 116.920,Y -36.935,Z -38.948,A -90.000,B 90.000,C 0.000} C_DIS
LIN {X 116.986,Y -21.308,Z -39.089,A -90.000,B 90.000,C 0.000} C_DIS
LIN {X 117.056,Y -21.308,Z -39.243,A -90.000,B 90.000,C 0.000} C_DIS
LIN {X 117.056,Y -60.000,Z -39.243,A -90.000,B 90.000,C 0.000} C_DIS
LIN {X 102.132,Y -60.000,Z -37.985,A -90.000,B 90.000,C 0.000} C_DIS
LIN {X 102.132,Y -21.308,Z -37.985,A -90.000,B 90.000,C 0.000} C_DIS
LIN {X 102.455,Y -21.308,Z -37.840,A -90.000,B 90.000,C 0.000} C_DIS
LIN {X 102.732,Y -21.308,Z -37.706,A -90.000,B 90.000,C 0.000} C_DIS
LIN {X 100.790,Y -21.307,Z -38.581,A -90.000,B 90.000,C 0.000} C_DIS
LIN {X 101.074,Y -21.308,Z -38.463,A -90.000,B 90.000,C 0.000} C_DIS
LIN {X 101.156,Y -21.308,Z -38.426,A -90.000,B 90.000,C 0.000} C_DIS
LIN {X 101.156,Y -60.000,Z -38.426,A -90.000,B 90.000,C 0.000} C_DIS
LIN {X 5.067,Y -60.000,Z -45.529,A -90.000,B 90.000,C 0.000} C_DIS
LIN {X 5.067,Y -21.308,Z -45.529,A -90.000,B 90.000,C 0.000} C_DIS
LIN {X 5.220,Y -21.333,Z -45.568,A -90.000,B 90.000,C 0.000} C_DIS
LIN {X 5.947,Y -21.440,Z -45.722,A -90.000,B 90.000,C 0.000} C_DIS
LIN {X 6.263,Y -21.490,Z -45.791,A -90.000,B 90.000,C 0.000} C_DIS
LIN {X 6.696,Y -21.567,Z -45.893,A -90.000,B 90.000,C 0.000} C_DIS
LIN {X 6.932,Y -21.607,Z -45.937,A -90.000,B 90.000,C 0.000} C_DIS
LIN {X 7.459,Y -21.694,Z -46.025,A -90.000,B 90.000,C 0.000} C_DIS
LIN {X 7.644,Y -21.726,Z -46.060,A -90.000,B 90.000,C 0.000} C_DIS
LIN {X 7.992,Y -21.789,Z -46.134,A -90.000,B 90.000,C 0.000} C_DIS
LIN {X 8.207,Y -21.831,Z -46.177,A -90.000,B 90.000,C 0.000} C_DIS
LIN {X 9.098,Y -21.995,Z -46.320,A -90.000,B 90.000,C 0.000} C_DIS
LIN {X 9.675,Y -22.106,Z -46.430,A -90.000,B 90.000,C 0.000} C_DIS
LIN {X 9.948,Y -22.161,Z -46.491,A -90.000,B 90.000,C 0.000} C_DIS
LIN {X 10.043,Y -22.146,Z -46.402,A -90.000,B 90.000,C 0.000} C_DIS
LIN {X 10.206,Y -22.121,Z -46.258,A -90.000,B 90.000,C 0.000} C_DIS
LIN {X 10.306,Y -22.110,Z -46.177,A -90.000,B 90.000,C 0.000} C_DIS
LIN {X 10.498,Y -22.093,Z -46.034,A -90.000,B 90.000,C 0.000} C_DIS
LIN {X 10.548,Y -22.089,Z -45.998,A -90.000,B 90.000,C 0.000} C_DIS
LIN {X 10.683,Y -22.059,Z -45.868,A -90.000,B 90.000,C 0.000} C_DIS
LIN {X 10.826,Y -22.030,Z -45.744,A -90.000,B 90.000,C 0.000} C_DIS
LIN {X 10.981,Y -22.002,Z -45.620,A -90.000,B 90.000,C 0.000} C_DIS
LIN {X 11.152,Y -21.977,Z -45.498,A -90.000,B 90.000,C 0.000} C_DIS
LIN {X 11.380,Y -21.933,Z -45.346,A -90.000,B 90.000,C 0.000} C_DIS
LIN {X 11.556,Y -21.904,Z -45.237,A -90.000,B 90.000,C 0.000} C_DIS
LIN {X 11.732,Y -21.876,Z -45.132,A -90.000,B 90.000,C 0.000} C_DIS
LIN {X 11.947,Y -21.838,Z -45.006,A -90.000,B 90.000,C 0.000} C_DIS
LIN {X 12.044,Y -21.818,Z -44.951,A -90.000,B 90.000,C 0.000} C_DIS
LIN {X 12.270,Y -21.761,Z -44.803,A -90.000,B 90.000,C 0.000} C_DIS
LIN {X 12.379,Y -21.737,Z -44.737,A -90.000,B 90.000,C 0.000} C_DIS
LIN {X 12.569,Y -21.697,Z -44.631,A -90.000,B 90.000,C 0.000} C_DIS
LIN {X 12.766,Y -21.662,Z -44.529,A -90.000,B 90.000,C 0.000} C_DIS
LIN {X 12.943,Y -21.630,Z -44.440,A -90.000,B 90.000,C 0.000} C_DIS
LIN {X 13.144,Y -21.599,Z -44.346,A -90.000,B 90.000,C 0.000} C_DIS
LIN {X 13.207,Y -21.587,Z -44.312,A -90.000,B 90.000,C 0.000} C_DIS
LIN {X 13.431,Y -21.530,Z -44.204,A -90.000,B 90.000,C 0.000} C_DIS
LIN {X 13.815,Y -21.438,Z -44.026,A -90.000,B 90.000,C 0.000} C_DIS
LIN {X 13.924,Y -21.414,Z -43.983,A -90.000,B 90.000,C 0.000} C_DIS
LIN {X 14.099,Y -21.373,Z -43.918,A -90.000,B 90.000,C 0.000} C_DIS
LIN {X 14.245,Y -21.341,Z -43.871,A -90.000,B 90.000,C 0.000} C_DIS
LIN {X 14.422,Y -21.308,Z -43.819,A -90.000,B 90.000,C 0.000} C_DIS
LIN {X 14.422,Y -60.000,Z -43.819,A -90.000,B 90.000,C 0.000} C_DIS
LIN {X -78.216,Y -60.000,Z -19.194,A -90.000,B 90.000,C 0.000} C_DIS
LIN {X -78.216,Y -21.308,Z -19.194,A -90.000,B 90.000,C 0.000} C_DIS
LIN {X -78.151,Y -21.310,Z -19.204,A -90.000,B 90.000,C 0.000} C_DIS
LIN {X -77.960,Y -21.319,Z -19.238,A -90.000,B 90.000,C 0.000} C_DIS
LIN {X -77.782,Y -21.327,Z -19.275,A -90.000,B 90.000,C 0.000} C_DIS
LIN {X -77.607,Y -21.333,Z -19.315,A -90.000,B 90.000,C 0.000} C_DIS
LIN {X -77.510,Y -21.335,Z -19.341,A -90.000,B 90.000,C 0.000} C_DIS
LIN {X -77.320,Y -21.343,Z -19.397,A -90.000,B 90.000,C 0.000} C_DIS
LIN {X -77.168,Y -21.348,Z -19.452,A -90.000,B 90.000,C 0.000} C_DIS
LIN {X -76.772,Y -21.371,Z -19.610,A -90.000,B 90.000,C 0.000} C_DIS
LIN {X -76.647,Y -21.382,Z -19.666,A -90.000,B 90.000,C 0.000} C_DIS
LIN {X -76.537,Y -21.395,Z -19.719,A -90.000,B 90.000,C 0.000} C_DIS
LIN {X -76.447,Y -21.402,Z -19.764,A -90.000,B 90.000,C 0.000} C_DIS
LIN {X -76.296,Y -21.409,Z -19.846,A -90.000,B 90.000,C 0.000} C_DIS
LIN {X -76.177,Y -21.419,Z -19.918,A -90.000,B 90.000,C 0.000} C_DIS
LIN {X -75.583,Y -21.472,Z -20.290,A -90.000,B 90.000,C 0.000} C_DIS
LIN {X -75.475,Y -21.479,Z -20.362,A -90.000,B 90.000,C 0.000} C_DIS
LIN {X -75.263,Y -21.493,Z -20.514,A -90.000,B 90.000,C 0.000} C_DIS
LIN {X -75.173,Y -21.502,Z -20.584,A -90.000,B 90.000,C 0.000} C_DIS
LIN {X -75.006,Y -21.524,Z -20.723,A -90.000,B 90.000,C 0.000} C_DIS
LIN {X -74.797,Y -21.555,Z -20.905,A -90.000,B 90.000,C 0.000} C_DIS
LIN {X -74.718,Y -21.566,Z -20.980,A -90.000,B 90.000,C 0.000} C_DIS
LIN {X -74.521,Y -21.592,Z -21.182,A -90.000,B 90.000,C 0.000} C_DIS
LIN {X -74.055,Y -21.669,Z -21.700,A -90.000,B 90.000,C 0.000} C_DIS
LIN {X -73.886,Y -21.697,Z -21.896,A -90.000,B 90.000,C 0.000} C_DIS
LIN {X -73.691,Y -21.680,Z -22.013,A -90.000,B 90.000,C 0.000} C_DIS
LIN {X -73.507,Y -21.670,Z -22.130,A -90.000,B 90.000,C 0.000} C_DIS
LIN {X -72.781,Y -21.639,Z -22.625,A -90.000,B 90.000,C 0.000} C_DIS
LIN {X -72.539,Y -21.623,Z -22.798,A -90.000,B 90.000,C 0.000} C_DIS
LIN {X -72.242,Y -21.607,Z -23.019,A -90.000,B 90.000,C 0.000} C_DIS
LIN {X -72.049,Y -21.603,Z -23.177,A -90.000,B 90.000,C 0.000} C_DIS
LIN {X -71.973,Y -21.603,Z -23.241,A -90.000,B 90.000,C 0.000} C_DIS
LIN {X -71.892,Y -21.604,Z -23.317,A -90.000,B 90.000,C 0.000} C_DIS
LIN {X -71.844,Y -21.605,Z -23.363,A -90.000,B 90.000,C 0.000} C_DIS
LIN {X -71.665,Y -21.603,Z -23.537,A -90.000,B 90.000,C 0.000} C_DIS
LIN {X -71.565,Y -21.601,Z -23.640,A -90.000,B 90.000,C 0.000} C_DIS
LIN {X -70.843,Y -21.577,Z -24.398,A -90.000,B 90.000,C 0.000} C_DIS
LIN {X -70.744,Y -21.575,Z -24.504,A -90.000,B 90.000,C 0.000} C_DIS
LIN {X -70.629,Y -21.569,Z -24.638,A -90.000,B 90.000,C 0.000} C_DIS
LIN {X -70.515,Y -21.566,Z -24.787,A -90.000,B 90.000,C 0.000} C_DIS
LIN {X -70.296,Y -21.553,Z -25.100,A -90.000,B 90.000,C 0.000} C_DIS
LIN {X -70.173,Y -21.550,Z -25.288,A -90.000,B 90.000,C 0.000} C_DIS
LIN {X -70.099,Y -21.552,Z -25.417,A -90.000,B 90.000,C 0.000} C_DIS
LIN {X -69.968,Y -21.560,Z -25.659,A -90.000,B 90.000,C 0.000} C_DIS
LIN {X -69.825,Y -21.575,Z -25.945,A -90.000,B 90.000,C 0.000} C_DIS
LIN {X -69.675,Y -21.586,Z -26.261,A -90.000,B 90.000,C 0.000} C_DIS
LIN {X -69.598,Y -21.580,Z -26.439,A -90.000,B 90.000,C 0.000} C_DIS
LIN {X -69.475,Y -21.563,Z -26.693,A -90.000,B 90.000,C 0.000} C_DIS
LIN {X -69.380,Y -21.548,Z -26.907,A -90.000,B 90.000,C 0.000} C_DIS
LIN {X -69.288,Y -21.531,Z -27.124,A -90.000,B 90.000,C 0.000} C_DIS
LIN {X -69.235,Y -21.523,Z -27.268,A -90.000,B 90.000,C 0.000} C_DIS
LIN {X -69.180,Y -21.517,Z -27.427,A -90.000,B 90.000,C 0.000} C_DIS
LIN {X -69.131,Y -21.515,Z -27.596,A -90.000,B 90.000,C 0.000} C_DIS
LIN {X -69.037,Y -21.514,Z -27.936,A -90.000,B 90.000,C 0.000} C_DIS
LIN {X -68.981,Y -21.514,Z -28.190,A -90.000,B 90.000,C 0.000} C_DIS
LIN {X -68.925,Y -21.512,Z -28.469,A -90.000,B 90.000,C 0.000} C_DIS
LIN {X -68.901,Y -21.514,Z -28.629,A -90.000,B 90.000,C 0.000} C_DIS
LIN {X -68.880,Y -21.518,Z -28.792,A -90.000,B 90.000,C 0.000} C_DIS
LIN {X -68.845,Y -21.528,Z -29.096,A -90.000,B 90.000,C 0.000} C_DIS
LIN {X -68.799,Y -21.536,Z -29.692,A -90.000,B 90.000,C 0.000} C_DIS
LIN {X -68.771,Y -21.551,Z -30.022,A -90.000,B 90.000,C 0.000} C_DIS
LIN {X -68.760,Y -21.563,Z -30.231,A -90.000,B 90.000,C 0.000} C_DIS
LIN {X -68.747,Y -21.596,Z -30.685,A -90.000,B 90.000,C 0.000} C_DIS
LIN {X -68.747,Y -21.620,Z -30.954,A -90.000,B 90.000,C 0.000} C_DIS
LIN {X -68.748,Y -21.635,Z -31.120,A -90.000,B 90.000,C 0.000} C_DIS
LIN {X -68.752,Y -21.652,Z -31.351,A -90.000,B 90.000,C 0.000} C_DIS
LIN {X -68.733,Y -21.815,Z -32.348,A -90.000,B 90.000,C 0.000} C_DIS
LIN {X -68.736,Y -21.838,Z -32.477,A -90.000,B 90.000,C 0.000} C_DIS
LIN {X -68.558,Y -21.783,Z -32.579,A -90.000,B 90.000,C 0.000} C_DIS
LIN {X -68.435,Y -21.768,Z -32.639,A -90.000,B 90.000,C 0.000} C_DIS
LIN {X -68.236,Y -21.739,Z -32.746,A -90.000,B 90.000,C 0.000} C_DIS
LIN {X -67.008,Y -21.571,Z -33.437,A -90.000,B 90.000,C 0.000} C_DIS
LIN {X -66.994,Y -21.570,Z -33.446,A -90.000,B 90.000,C 0.000} C_DIS
LIN {X -66.384,Y -21.555,Z -33.783,A -90.000,B 90.000,C 0.000} C_DIS
LIN {X -65.960,Y -21.539,Z -34.018,A -90.000,B 90.000,C 0.000} C_DIS
LIN {X -64.977,Y -21.490,Z -34.532,A -90.000,B 90.000,C 0.000} C_DIS
LIN {X -64.036,Y -21.482,Z -35.003,A -90.000,B 90.000,C 0.000} C_DIS
LIN {X -63.583,Y -21.483,Z -35.244,A -90.000,B 90.000,C 0.000} C_DIS
LIN {X -62.618,Y -21.464,Z -35.708,A -90.000,B 90.000,C 0.000} C_DIS
LIN {X -61.349,Y -21.469,Z -36.303,A -90.000,B 90.000,C 0.000} C_DIS
LIN {X -61.106,Y -21.472,Z -36.421,A -90.000,B 90.000,C 0.000} C_DIS
LIN {X -60.078,Y -21.465,Z -36.870,A -90.000,B 90.000,C 0.000} C_DIS
LIN {X -59.358,Y -21.468,Z -37.180,A -90.000,B 90.000,C 0.000} C_DIS
LIN {X -58.576,Y -21.472,Z -37.517,A -90.000,B 90.000,C 0.000} C_DIS
LIN {X -57.832,Y -21.462,Z -37.805,A -90.000,B 90.000,C 0.000} C_DIS
LIN {X -56.211,Y -21.465,Z -38.421,A -90.000,B 90.000,C 0.000} C_DIS
LIN {X -55.132,Y -21.451,Z -38.785,A -90.000,B 90.000,C 0.000} C_DIS
LIN {X -53.515,Y -21.452,Z -39.323,A -90.000,B 90.000,C 0.000} C_DIS
LIN {X -53.034,Y -21.449,Z -39.474,A -90.000,B 90.000,C 0.000} C_DIS
LIN {X -52.432,Y -21.441,Z -39.653,A -90.000,B 90.000,C 0.000} C_DIS
LIN {X -50.847,Y -21.453,Z -40.110,A -90.000,B 90.000,C 0.000} C_DIS
LIN {X -49.511,Y -21.455,Z -40.470,A -90.000,B 90.000,C 0.000} C_DIS
LIN {X -49.090,Y -21.458,Z -40.582,A -90.000,B 90.000,C 0.000} C_DIS
LIN {X -48.320,Y -21.460,Z -40.777,A -90.000,B 90.000,C 0.000} C_DIS
LIN {X -48.100,Y -21.463,Z -40.831,A -90.000,B 90.000,C 0.000} C_DIS
LIN {X -47.569,Y -21.465,Z -40.948,A -90.000,B 90.000,C 0.000} C_DIS
LIN {X -46.631,Y -21.474,Z -41.169,A -90.000,B 90.000,C 0.000} C_DIS
LIN {X -45.993,Y -21.475,Z -41.310,A -90.000,B 90.000,C 0.000} C_DIS
LIN {X -45.542,Y -21.493,Z -41.402,A -90.000,B 90.000,C 0.000} C_DIS
LIN {X -45.143,Y -21.511,Z -41.495,A -90.000,B 90.000,C 0.000} C_DIS
LIN {X -45.080,Y -21.514,Z -41.507,A -90.000,B 90.000,C 0.000} C_DIS
LIN {X -44.356,Y -21.604,Z -41.623,A -90.000,B 90.000,C 0.000} C_DIS
LIN {X -43.910,Y -21.665,Z -41.696,A -90.000,B 90.000,C 0.000} C_DIS
LIN {X -43.507,Y -21.720,Z -41.771,A -90.000,B 90.000,C 0.000} C_DIS
LIN {X -43.317,Y -21.757,Z -41.808,A -90.000,B 90.000,C 0.000} C_DIS
LIN {X -42.752,Y -21.865,Z -41.922,A -90.000,B 90.000,C 0.000} C_DIS
LIN {X -42.297,Y -21.945,Z -42.023,A -90.000,B 90.000,C 0.000} C_DIS
LIN {X -41.913,Y -22.006,Z -42.111,A -90.000,B 90.000,C 0.000} C_DIS
LIN {X -41.759,Y -22.031,Z -42.144,A -90.000,B 90.000,C 0.000} C_DIS
LIN {X -41.427,Y -22.093,Z -42.218,A -90.000,B 90.000,C 0.000} C_DIS
LIN {X -41.316,Y -22.111,Z -42.246,A -90.000,B 90.000,C 0.000} C_DIS
LIN {X -40.758,Y -22.192,Z -42.387,A -90.000,B 90.000,C 0.000} C_DIS
LIN {X -40.334,Y -22.251,Z -42.463,A -90.000,B 90.000,C 0.000} C_DIS
LIN {X -39.566,Y -22.390,Z -42.601,A -90.000,B 90.000,C 0.000} C_DIS
LIN {X -39.372,Y -22.425,Z -42.634,A -90.000,B 90.000,C 0.000} C_DIS
LIN {X -38.885,Y -22.506,Z -42.719,A -90.000,B 90.000,C 0.000} C_DIS
LIN {X -38.691,Y -22.535,Z -42.755,A -90.000,B 90.000,C 0.000} C_DIS
LIN {X -38.447,Y -22.572,Z -42.810,A -90.000,B 90.000,C 0.000} C_DIS
LIN {X -37.873,Y -22.654,Z -42.945,A -90.000,B 90.000,C 0.000} C_DIS
LIN {X -37.390,Y -22.712,Z -43.067,A -90.000,B 90.000,C 0.000} C_DIS
LIN {X -36.660,Y -22.792,Z -43.257,A -90.000,B 90.000,C 0.000} C_DIS
LIN {X -35.840,Y -22.882,Z -43.474,A -90.000,B 90.000,C 0.000} C_DIS
LIN {X -35.762,Y -22.877,Z -43.372,A -90.000,B 90.000,C 0.000} C_DIS
LIN {X -35.655,Y -22.872,Z -43.248,A -90.000,B 90.000,C 0.000} C_DIS
LIN {X -35.518,Y -22.866,Z -43.102,A -90.000,B 90.000,C 0.000} C_DIS
LIN {X -35.354,Y -22.857,Z -42.936,A -90.000,B 90.000,C 0.000} C_DIS
LIN {X -35.210,Y -22.848,Z -42.803,A -90.000,B 90.000,C 0.000} C_DIS
LIN {X -35.046,Y -22.841,Z -42.667,A -90.000,B 90.000,C 0.000} C_DIS
LIN {X -34.940,Y -22.833,Z -42.583,A -90.000,B 90.000,C 0.000} C_DIS
LIN {X -34.820,Y -22.826,Z -42.494,A -90.000,B 90.000,C 0.000} C_DIS
LIN {X -34.727,Y -22.820,Z -42.425,A -90.000,B 90.000,C 0.000} C_DIS
LIN {X -34.590,Y -22.805,Z -42.325,A -90.000,B 90.000,C 0.000} C_DIS
LIN {X -34.313,Y -22.759,Z -42.127,A -90.000,B 90.000,C 0.000} C_DIS
LIN {X -34.136,Y -22.730,Z -42.007,A -90.000,B 90.000,C 0.000} C_DIS
LIN {X -34.048,Y -22.716,Z -41.951,A -90.000,B 90.000,C 0.000} C_DIS
LIN {X -32.935,Y -22.561,Z -41.303,A -90.000,B 90.000,C 0.000} C_DIS
LIN {X -32.688,Y -22.528,Z -41.168,A -90.000,B 90.000,C 0.000} C_DIS
LIN {X -32.571,Y -22.512,Z -41.114,A -90.000,B 90.000,C 0.000} C_DIS
LIN {X -32.198,Y -22.465,Z -40.954,A -90.000,B 90.000,C 0.000} C_DIS
LIN {X -32.151,Y -22.460,Z -40.936,A -90.000,B 90.000,C 0.000} C_DIS
LIN {X -32.002,Y -22.440,Z -40.888,A -90.000,B 90.000,C 0.000} C_DIS
LIN {X -31.898,Y -22.429,Z -40.860,A -90.000,B 90.000,C 0.000} C_DIS
LIN {X -31.633,Y -22.402,Z -40.795,A -90.000,B 90.000,C 0.000} C_DIS
LIN {X -31.406,Y -22.381,Z -40.747,A -90.000,B 90.000,C 0.000} C_DIS
LIN {X -31.268,Y -22.372,Z -40.728,A -90.000,B 90.000,C 0.000} C_DIS
LIN {X -30.858,Y -22.349,Z -40.683,A -90.000,B 90.000,C 0.000} C_DIS
LIN {X -30.738,Y -22.347,Z -40.682,A -90.000,B 90.000,C 0.000} C_DIS
LIN {X -30.532,Y -22.342,Z -40.675,A -90.000,B 90.000,C 0.000} C_DIS
LIN {X -29.008,Y -22.327,Z -40.701,A -90.000,B 90.000,C 0.000} C_DIS
LIN {X -28.768,Y -22.324,Z -40.708,A -90.000,B 90.000,C 0.000} C_DIS
LIN {X -28.271,Y -22.308,Z -40.700,A -90.000,B 90.000,C 0.000} C_DIS
LIN {X -27.702,Y -22.299,Z -40.691,A -90.000,B 90.000,C 0.000} C_DIS
LIN {X -27.533,Y -22.295,Z -40.690,A -90.000,B 90.000,C 0.000} C_DIS
LIN {X -27.059,Y -22.277,Z -40.686,A -90.000,B 90.000,C 0.000} C_DIS
LIN {X -26.950,Y -22.274,Z -40.688,A -90.000,B 90.000,C 0.000} C_DIS
LIN {X -26.569,Y -22.267,Z -40.705,A -90.000,B 90.000,C 0.000} C_DIS
LIN {X -26.282,Y -22.244,Z -40.672,A -90.000,B 90.000,C 0.000} C_DIS
LIN {X -26.194,Y -22.238,Z -40.664,A -90.000,B 90.000,C 0.000} C_DIS
LIN {X -25.972,Y -22.224,Z -40.648,A -90.000,B 90.000,C 0.000} C_DIS
LIN {X -25.053,Y -22.202,Z -40.585,A -90.000,B 90.000,C 0.000} C_DIS
LIN {X -24.846,Y -22.200,Z -40.578,A -90.000,B 90.000,C 0.000} C_DIS
LIN {X -24.704,Y -22.200,Z -40.577,A -90.000,B 90.000,C 0.000} C_DIS
LIN {X -24.512,Y -22.200,Z -40.577,A -90.000,B 90.000,C 0.000} C_DIS
LIN {X -24.411,Y -22.200,Z -40.579,A -90.000,B 90.000,C 0.000} C_DIS
LIN {X -24.237,Y -22.192,Z -40.564,A -90.000,B 90.000,C 0.000} C_DIS
LIN {X -23.846,Y -22.181,Z -40.547,A -90.000,B 90.000,C 0.000} C_DIS
LIN {X -23.124,Y -22.179,Z -40.511,A -90.000,B 90.000,C 0.000} C_DIS
LIN {X -22.588,Y -22.165,Z -40.489,A -90.000,B 90.000,C 0.000} C_DIS
LIN {X -22.109,Y -22.133,Z -40.425,A -90.000,B 90.000,C 0.000} C_DIS
LIN {X -21.517,Y -22.091,Z -40.348,A -90.000,B 90.000,C 0.000} C_DIS
LIN {X -20.868,Y -22.051,Z -40.262,A -90.000,B 90.000,C 0.000} C_DIS
LIN {X -20.524,Y -22.036,Z -40.232,A -90.000,B 90.000,C 0.000} C_DIS
LIN {X -20.409,Y -22.032,Z -40.226,A -90.000,B 90.000,C 0.000} C_DIS
LIN {X -20.030,Y -22.026,Z -40.216,A -90.000,B 90.000,C 0.000} C_DIS
LIN {X -19.485,Y -22.012,Z -40.196,A -90.000,B 90.000,C 0.000} C_DIS
LIN {X -19.019,Y -22.002,Z -40.184,A -90.000,B 90.000,C 0.000} C_DIS
LIN {X -18.194,Y -21.977,Z -40.164,A -90.000,B 90.000,C 0.000} C_DIS
LIN {X -18.022,Y -21.969,Z -40.161,A -90.000,B 90.000,C 0.000} C_DIS
LIN {X -17.296,Y -21.919,Z -40.156,A -90.000,B 90.000,C 0.000} C_DIS
LIN {X -16.853,Y -21.894,Z -40.162,A -90.000,B 90.000,C 0.000} C_DIS
LIN {X -15.966,Y -21.836,Z -40.175,A -90.000,B 90.000,C 0.000} C_DIS
LIN {X -14.778,Y -21.740,Z -40.202,A -90.000,B 90.000,C 0.000} C_DIS
LIN {X -14.034,Y -21.694,Z -40.233,A -90.000,B 90.000,C 0.000} C_DIS
LIN {X -13.874,Y -21.687,Z -40.244,A -90.000,B 90.000,C 0.000} C_DIS
LIN {X -13.493,Y -21.673,Z -40.277,A -90.000,B 90.000,C 0.000} C_DIS
LIN {X -12.741,Y -21.623,Z -40.355,A -90.000,B 90.000,C 0.000} C_DIS
LIN {X -12.456,Y -21.608,Z -40.393,A -90.000,B 90.000,C 0.000} C_DIS
LIN {X -11.820,Y -21.570,Z -40.485,A -90.000,B 90.000,C 0.000} C_DIS
LIN {X -10.978,Y -21.508,Z -40.615,A -90.000,B 90.000,C 0.000} C_DIS
LIN {X -10.307,Y -21.462,Z -40.721,A -90.000,B 90.000,C 0.000} C_DIS
LIN {X -9.201,Y -21.414,Z -40.924,A -90.000,B 90.000,C 0.000} C_DIS
LIN {X -8.766,Y -21.387,Z -41.009,A -90.000,B 90.000,C 0.000} C_DIS
LIN {X -8.651,Y -21.381,Z -41.033,A -90.000,B 90.000,C 0.000} C_DIS
LIN {X -7.554,Y -21.308,Z -41.276,A -90.000,B 90.000,C 0.000} C_DIS
LIN {X -7.554,Y -60.000,Z -41.276,A -90.000,B 90.000,C 0.000} C_DIS
LIN {X -44.674,Y -60.000,Z -39.559,A -90.000,B 90.000,C 0.000} C_DIS
LIN {X -44.674,Y -21.308,Z -39.559,A -90.000,B 90.000,C 0.000} C_DIS
LIN {X -44.017,Y -21.397,Z -39.663,A -90.000,B 90.000,C 0.000} C_DIS
LIN {X -43.638,Y -21.468,Z -39.723,A -90.000,B 90.000,C 0.000} C_DIS
LIN {X -43.420,Y -21.506,Z -39.761,A -90.000,B 90.000,C 0.000} C_DIS
LIN {X -43.079,Y -21.565,Z -39.823,A -90.000,B 90.000,C 0.000} C_DIS
LIN {X -42.445,Y -21.667,Z -39.952,A -90.000,B 90.000,C 0.000} C_DIS
LIN {X -42.292,Y -21.689,Z -39.984,A -90.000,B 90.000,C 0.000} C_DIS
LIN {X -41.929,Y -21.742,Z -40.065,A -90.000,B 90.000,C 0.000} C_DIS
LIN {X -41.596,Y -21.784,Z -40.142,A -90.000,B 90.000,C 0.000} C_DIS
LIN {X -41.232,Y -21.846,Z -40.223,A -90.000,B 90.000,C 0.000} C_DIS
LIN {X -40.980,Y -21.881,Z -40.280,A -90.000,B 90.000,C 0.000} C_DIS
LIN {X -40.309,Y -21.968,Z -40.450,A -90.000,B 90.000,C 0.000} C_DIS
LIN {X -39.889,Y -22.016,Z -40.526,A -90.000,B 90.000,C 0.000} C_DIS
LIN {X -38.992,Y -22.156,Z -40.689,A -90.000,B 90.000,C 0.000} C_DIS
LIN {X -38.277,Y -22.267,Z -40.817,A -90.000,B 90.000,C 0.000} C_DIS
LIN {X -37.642,Y -22.360,Z -40.962,A -90.000,B 90.000,C 0.000} C_DIS
LIN {X -37.357,Y -22.389,Z -41.031,A -90.000,B 90.000,C 0.000} C_DIS
LIN {X -37.075,Y -22.418,Z -41.103,A -90.000,B 90.000,C 0.000} C_DIS
LIN {X -36.769,Y -22.448,Z -41.182,A -90.000,B 90.000,C 0.000} C_DIS
LIN {X -36.439,Y -22.479,Z -41.268,A -90.000,B 90.000,C 0.000} C_DIS
LIN {X -36.218,Y -22.438,Z -41.095,A -90.000,B 90.000,C 0.000} C_DIS
LIN {X -36.120,Y -22.421,Z -41.022,A -90.000,B 90.000,C 0.000} C_DIS
LIN {X -35.778,Y -22.364,Z -40.778,A -90.000,B 90.000,C 0.000} C_DIS
LIN {X -35.436,Y -22.301,Z -40.536,A -90.000,B 90.000,C 0.000} C_DIS
LIN {X -35.219,Y -22.264,Z -40.391,A -90.000,B 90.000,C 0.000} C_DIS
LIN {X -35.083,Y -22.242,Z -40.307,A -90.000,B 90.000,C 0.000} C_DIS
LIN {X -34.413,Y -22.141,Z -39.919,A -90.000,B 90.000,C 0.000} C_DIS
LIN {X -33.909,Y -22.031,Z -39.638,A -90.000,B 90.000,C 0.000} C_DIS
LIN {X -33.595,Y -21.966,Z -39.477,A -90.000,B 90.000,C 0.000} C_DIS
LIN {X -33.383,Y -21.928,Z -39.381,A -90.000,B 90.000,C 0.000} C_DIS
LIN {X -33.011,Y -21.866,Z -39.228,A -90.000,B 90.000,C 0.000} C_DIS
